ABB RAPID module: d6a8df4c.mod

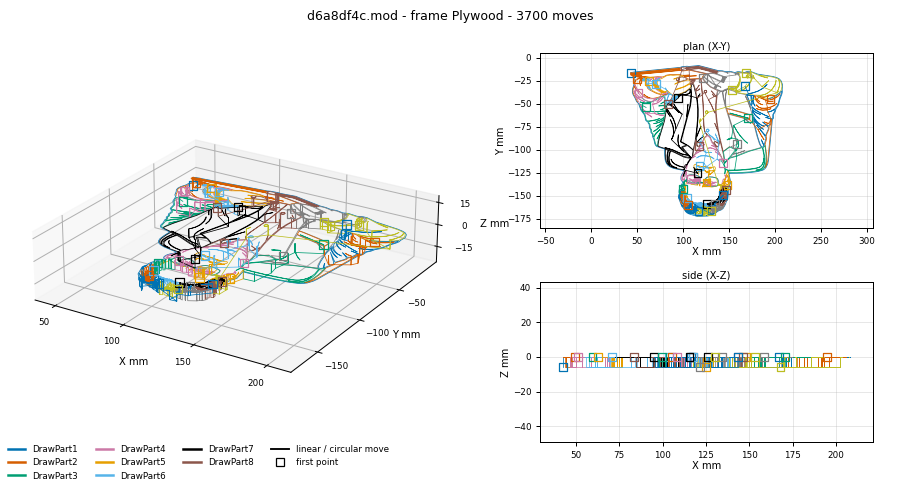
[picture p0: tool path of d6a8df4c.mod in frame Plywood, 3700 of 3702 moves have a stored position in this frame; points joined in program order, loops and branches not executed]
MODULE ImageDraw
  ! Generated 2026-10-07 09:12 for ABB GoFa CRB 15000-5/0.95: 203 strokes
  ! Page 250 x 180 mm. Work object Plywood: Z points DOWN, so pen-up is -Z and the tool uses orientation [1,0,0,0].
  ! Uses the tool 'tcp' and work object 'Plywood' that already exist on the controller.
  CONST robtarget pOrigin:=[[0,0,0],[1,0,0,0],[0,0,0,0],[9E9,9E9,9E9,9E9,9E9,9E9]];
  CONST jointtarget jHome:=[[0,0,0,0,30,0],[9E9,9E9,9E9,9E9,9E9,9E9]];
  CONST speeddata vTravel:=[250,200,5000,1000];

  PROC DrawImage()
    SingArea\Wrist;
    ConfL\Off;
    ConfJ\Off;
    MoveAbsJ jHome\NoEOffs,vTravel,fine,tcp;
    DrawPart1;
    DrawPart2;
    DrawPart3;
    DrawPart4;
    DrawPart5;
    DrawPart6;
    DrawPart7;
    DrawPart8;
    DrawPart9;
    DrawPart10;
    DrawPart11;
    DrawPart12;
    DrawPart13;
    DrawPart14;
    DrawPart15;
    DrawPart16;
    DrawPart17;
    DrawPart18;
    DrawPart19;
    DrawPart20;
    DrawPart21;
    DrawPart22;
    DrawPart23;
    DrawPart24;
    DrawPart25;
    DrawPart26;
    DrawPart27;
    DrawPart28;
    DrawPart29;
    DrawPart30;
    DrawPart31;
    MoveAbsJ jHome\NoEOffs,vTravel,fine,tcp;
  ENDPROC

  PROC DrawPart1()
    MoveL Offs(pOrigin,42.73,-16.05,-6.00),vTravel,z5,tcp\WObj:=Plywood;
    MoveL Offs(pOrigin,42.73,-16.05,-0.00),v60,z0,tcp\WObj:=Plywood;
    MoveL Offs(pOrigin,46.16,-15.41,-0.00),v40,z0,tcp\WObj:=Plywood;
    MoveL Offs(pOrigin,96.63,-10.31,-0.00),v40,z0,tcp\WObj:=Plywood;
    MoveL Offs(pOrigin,98.76,-9.57,-0.00),v40,z0,tcp\WObj:=Plywood;
    MoveL Offs(pOrigin,104.18,-9.04,-0.00),v40,z0,tcp\WObj:=Plywood;
    MoveL Offs(pOrigin,106.09,-9.36,-0.00),v40,z0,tcp\WObj:=Plywood;
    MoveL Offs(pOrigin,116.93,-8.29,-0.00),v40,z0,tcp\WObj:=Plywood;
    MoveL Offs(pOrigin,138.28,-13.82,-0.00),v40,z0,tcp\WObj:=Plywood;
    MoveL Offs(pOrigin,142.64,-14.03,-0.00),v40,z0,tcp\WObj:=Plywood;
    MoveL Offs(pOrigin,146.36,-14.99,-0.00),v40,z0,tcp\WObj:=Plywood;
    MoveL Offs(pOrigin,151.77,-14.77,-0.00),v40,z0,tcp\WObj:=Plywood;
    MoveL Offs(pOrigin,156.24,-15.94,-0.00),v40,z0,tcp\WObj:=Plywood;
    MoveL Offs(pOrigin,159.11,-14.99,-0.00),v40,z0,tcp\WObj:=Plywood;
    MoveL Offs(pOrigin,160.81,-14.99,-0.00),v40,z0,tcp\WObj:=Plywood;
    MoveL Offs(pOrigin,166.54,-15.94,-0.00),v40,z0,tcp\WObj:=Plywood;
    MoveL Offs(pOrigin,170.26,-14.56,-0.00),v40,z0,tcp\WObj:=Plywood;
    MoveL Offs(pOrigin,173.02,-14.56,-0.00),v40,z0,tcp\WObj:=Plywood;
    MoveL Offs(pOrigin,181.10,-17.64,-0.00),v40,z0,tcp\WObj:=Plywood;
    MoveL Offs(pOrigin,197.99,-20.30,-0.00),v40,z0,tcp\WObj:=Plywood;
    MoveL Offs(pOrigin,202.14,-21.54,-0.00),v40,z0,tcp\WObj:=Plywood;
    MoveL Offs(pOrigin,204.79,-22.96,-0.00),v40,z0,tcp\WObj:=Plywood;
    MoveL Offs(pOrigin,206.74,-25.19,-0.00),v40,z0,tcp\WObj:=Plywood;
    MoveL Offs(pOrigin,207.98,-28.59,-0.00),v40,z0,tcp\WObj:=Plywood;
    MoveL Offs(pOrigin,208.19,-30.08,-0.00),v40,z0,tcp\WObj:=Plywood;
    MoveL Offs(pOrigin,207.77,-34.33,-0.00),v40,z0,tcp\WObj:=Plywood;
    MoveL Offs(pOrigin,207.98,-37.09,-0.00),v40,z0,tcp\WObj:=Plywood;
    MoveL Offs(pOrigin,207.38,-39.64,-0.00),v40,z0,tcp\WObj:=Plywood;
    MoveL Offs(pOrigin,205.54,-44.31,-0.00),v40,z0,tcp\WObj:=Plywood;
    MoveL Offs(pOrigin,203.77,-51.01,-0.00),v40,z0,tcp\WObj:=Plywood;
    MoveL Offs(pOrigin,203.06,-52.60,-0.00),v40,z0,tcp\WObj:=Plywood;
    MoveL Offs(pOrigin,201.15,-55.26,-0.00),v40,z0,tcp\WObj:=Plywood;
    MoveL Offs(pOrigin,200.15,-58.66,-0.00),v40,z0,tcp\WObj:=Plywood;
    MoveL Offs(pOrigin,198.49,-61.31,-0.00),v40,z0,tcp\WObj:=Plywood;
    MoveL Offs(pOrigin,198.42,-65.14,-0.00),v40,z0,tcp\WObj:=Plywood;
    MoveL Offs(pOrigin,197.89,-66.31,-0.00),v40,z0,tcp\WObj:=Plywood;
    MoveL Offs(pOrigin,197.14,-66.94,-0.00),v40,z0,tcp\WObj:=Plywood;
    MoveL Offs(pOrigin,192.89,-111.36,-0.00),v40,z0,tcp\WObj:=Plywood;
    MoveL Offs(pOrigin,192.15,-115.18,-0.00),v40,z0,tcp\WObj:=Plywood;
    MoveL Offs(pOrigin,190.45,-119.01,-0.00),v40,z0,tcp\WObj:=Plywood;
    MoveL Offs(pOrigin,188.75,-120.92,-0.00),v40,z0,tcp\WObj:=Plywood;
    MoveL Offs(pOrigin,186.73,-122.23,-0.00),v40,z0,tcp\WObj:=Plywood;
    MoveL Offs(pOrigin,181.10,-123.79,-0.00),v40,z0,tcp\WObj:=Plywood;
    MoveL Offs(pOrigin,173.88,-124.74,-0.00),v40,z0,tcp\WObj:=Plywood;
    MoveL Offs(pOrigin,164.31,-125.49,-0.00),v40,z0,tcp\WObj:=Plywood;
    MoveL Offs(pOrigin,149.76,-125.74,-0.00),v40,z0,tcp\WObj:=Plywood;
    MoveL Offs(pOrigin,151.67,-135.16,-0.00),v40,z0,tcp\WObj:=Plywood;
    MoveL Offs(pOrigin,151.07,-137.60,-0.00),v40,z0,tcp\WObj:=Plywood;
    MoveL Offs(pOrigin,150.00,-139.41,-0.00),v40,z0,tcp\WObj:=Plywood;
    MoveL Offs(pOrigin,150.15,-140.26,-0.00),v40,z0,tcp\WObj:=Plywood;
    MoveL Offs(pOrigin,149.76,-140.79,-0.00),v40,z0,tcp\WObj:=Plywood;
    MoveL Offs(pOrigin,149.44,-143.55,-0.00),v40,z0,tcp\WObj:=Plywood;
    MoveL Offs(pOrigin,149.12,-143.76,-0.00),v40,z0,tcp\WObj:=Plywood;
    MoveL Offs(pOrigin,149.23,-147.27,-0.00),v40,z0,tcp\WObj:=Plywood;
    MoveL Offs(pOrigin,148.23,-154.81,-0.00),v40,z0,tcp\WObj:=Plywood;
    MoveL Offs(pOrigin,147.03,-156.19,-0.00),v40,z0,tcp\WObj:=Plywood;
    MoveL Offs(pOrigin,146.11,-159.38,-0.00),v40,z0,tcp\WObj:=Plywood;
    MoveL Offs(pOrigin,143.49,-163.95,-0.00),v40,z0,tcp\WObj:=Plywood;
    MoveL Offs(pOrigin,141.57,-165.47,-0.00),v40,z0,tcp\WObj:=Plywood;
    MoveL Offs(pOrigin,137.86,-166.89,-0.00),v40,z0,tcp\WObj:=Plywood;
    MoveL Offs(pOrigin,134.14,-169.83,-0.00),v40,z0,tcp\WObj:=Plywood;
    MoveL Offs(pOrigin,132.12,-170.75,-0.00),v40,z0,tcp\WObj:=Plywood;
    MoveL Offs(pOrigin,126.38,-172.24,-0.00),v40,z0,tcp\WObj:=Plywood;
    MoveL Offs(pOrigin,115.22,-172.56,-0.00),v40,z0,tcp\WObj:=Plywood;
    MoveL Offs(pOrigin,106.41,-169.94,-0.00),v40,z0,tcp\WObj:=Plywood;
    MoveL Offs(pOrigin,104.18,-168.84,-0.00),v40,z0,tcp\WObj:=Plywood;
    MoveL Offs(pOrigin,102.58,-167.35,-0.00),v40,z0,tcp\WObj:=Plywood;
    MoveL Offs(pOrigin,100.67,-164.06,-0.00),v40,z0,tcp\WObj:=Plywood;
    MoveL Offs(pOrigin,98.30,-161.40,-0.00),v40,z0,tcp\WObj:=Plywood;
    MoveL Offs(pOrigin,94.72,-151.73,-0.00),v40,z0,tcp\WObj:=Plywood;
    MoveL Offs(pOrigin,94.93,-149.61,-0.00),v40,z0,tcp\WObj:=Plywood;
    MoveL Offs(pOrigin,95.75,-147.80,-0.00),v40,z0,tcp\WObj:=Plywood;
    MoveL Offs(pOrigin,95.36,-146.21,-0.00),v40,z0,tcp\WObj:=Plywood;
    MoveL Offs(pOrigin,95.57,-143.76,-0.00),v40,z0,tcp\WObj:=Plywood;
    MoveL Offs(pOrigin,96.60,-140.68,-0.00),v40,z0,tcp\WObj:=Plywood;
    MoveL Offs(pOrigin,99.50,-135.58,-0.00),v40,z0,tcp\WObj:=Plywood;
    MoveL Offs(pOrigin,99.50,-134.73,-0.00),v40,z0,tcp\WObj:=Plywood;
    MoveL Offs(pOrigin,98.65,-134.31,-0.00),v40,z0,tcp\WObj:=Plywood;
    MoveL Offs(pOrigin,97.80,-133.14,-0.00),v40,z0,tcp\WObj:=Plywood;
    MoveL Offs(pOrigin,97.48,-131.76,-0.00),v40,z0,tcp\WObj:=Plywood;
    MoveL Offs(pOrigin,97.59,-129.10,-0.00),v40,z0,tcp\WObj:=Plywood;
    MoveL Offs(pOrigin,98.19,-127.51,-0.00),v40,z0,tcp\WObj:=Plywood;
    MoveL Offs(pOrigin,99.68,-125.17,-0.00),v40,z0,tcp\WObj:=Plywood;
    MoveL Offs(pOrigin,100.53,-122.72,-0.00),v40,z0,tcp\WObj:=Plywood;
    MoveL Offs(pOrigin,89.51,-120.28,-0.00),v40,z0,tcp\WObj:=Plywood;
    MoveL Offs(pOrigin,85.58,-118.62,-0.00),v40,z0,tcp\WObj:=Plywood;
    MoveL Offs(pOrigin,83.46,-117.09,-0.00),v40,z0,tcp\WObj:=Plywood;
    MoveL Offs(pOrigin,81.61,-114.76,-0.00),v40,z0,tcp\WObj:=Plywood;
    MoveL Offs(pOrigin,80.38,-111.46,-0.00),v40,z0,tcp\WObj:=Plywood;
    MoveL Offs(pOrigin,79.84,-106.26,-0.00),v40,z0,tcp\WObj:=Plywood;
    MoveL Offs(pOrigin,79.77,-99.24,-0.00),v40,z0,tcp\WObj:=Plywood;
    MoveL Offs(pOrigin,71.66,-96.62,-0.00),v40,z0,tcp\WObj:=Plywood;
    MoveL Offs(pOrigin,70.71,-96.06,-0.00),v40,z0,tcp\WObj:=Plywood;
    MoveL Offs(pOrigin,69.61,-94.68,-0.00),v40,z0,tcp\WObj:=Plywood;
    MoveL Offs(pOrigin,68.90,-92.97,-0.00),v40,z0,tcp\WObj:=Plywood;
    MoveL Offs(pOrigin,68.16,-89.26,-0.00),v40,z0,tcp\WObj:=Plywood;
    MoveL Offs(pOrigin,66.56,-85.43,-0.00),v40,z0,tcp\WObj:=Plywood;
    MoveL Offs(pOrigin,66.39,-82.99,-0.00),v40,z0,tcp\WObj:=Plywood;
    MoveL Offs(pOrigin,64.86,-81.07,-0.00),v40,z0,tcp\WObj:=Plywood;
    MoveL Offs(pOrigin,64.69,-77.99,-0.00),v40,z0,tcp\WObj:=Plywood;
    MoveL Offs(pOrigin,63.69,-76.93,-0.00),v40,z0,tcp\WObj:=Plywood;
    MoveL Offs(pOrigin,63.16,-75.76,-0.00),v40,z0,tcp\WObj:=Plywood;
    MoveL Offs(pOrigin,62.99,-72.47,-0.00),v40,z0,tcp\WObj:=Plywood;
    MoveL Offs(pOrigin,61.82,-70.88,-0.00),v40,z0,tcp\WObj:=Plywood;
    MoveL Offs(pOrigin,61.46,-69.39,-0.00),v40,z0,tcp\WObj:=Plywood;
    MoveL Offs(pOrigin,60.19,-69.00,-0.00),v40,z0,tcp\WObj:=Plywood;
    MoveL Offs(pOrigin,59.20,-68.01,-0.00),v40,z0,tcp\WObj:=Plywood;
    MoveL Offs(pOrigin,57.89,-62.27,-0.00),v40,z0,tcp\WObj:=Plywood;
    MoveL Offs(pOrigin,53.88,-56.85,-0.00),v40,z0,tcp\WObj:=Plywood;
    MoveL Offs(pOrigin,51.33,-49.62,-0.00),v40,z0,tcp\WObj:=Plywood;
    MoveL Offs(pOrigin,49.78,-48.24,-0.00),v40,z0,tcp\WObj:=Plywood;
    MoveL Offs(pOrigin,49.00,-47.08,-0.00),v40,z0,tcp\WObj:=Plywood;
    MoveL Offs(pOrigin,47.15,-42.93,-0.00),v40,z0,tcp\WObj:=Plywood;
    MoveL Offs(pOrigin,45.49,-40.17,-0.00),v40,z0,tcp\WObj:=Plywood;
    MoveL Offs(pOrigin,44.67,-37.51,-0.00),v40,z0,tcp\WObj:=Plywood;
    MoveL Offs(pOrigin,44.78,-34.11,-0.00),v40,z0,tcp\WObj:=Plywood;
    MoveL Offs(pOrigin,46.27,-29.23,-0.00),v40,z0,tcp\WObj:=Plywood;
    MoveL Offs(pOrigin,46.16,-27.42,-0.00),v40,z0,tcp\WObj:=Plywood;
    MoveL Offs(pOrigin,46.66,-25.51,-0.00),v40,z0,tcp\WObj:=Plywood;
    MoveL Offs(pOrigin,48.08,-23.81,-0.00),v40,z0,tcp\WObj:=Plywood;
  ENDPROC

  PROC DrawPart2()
    MoveL Offs(pOrigin,49.56,-22.89,-0.00),v40,z0,tcp\WObj:=Plywood;
    MoveL Offs(pOrigin,54.10,-21.68,-0.00),v40,z0,tcp\WObj:=Plywood;
    MoveL Offs(pOrigin,43.29,-19.06,-0.00),v40,z0,tcp\WObj:=Plywood;
    MoveL Offs(pOrigin,42.55,-18.17,-0.00),v40,z0,tcp\WObj:=Plywood;
    MoveL Offs(pOrigin,42.73,-16.05,-0.00),v40,z0,tcp\WObj:=Plywood;
    MoveL Offs(pOrigin,43.51,-16.40,-0.00),v40,z0,tcp\WObj:=Plywood;
    MoveL Offs(pOrigin,43.22,-17.01,-0.00),v40,z0,tcp\WObj:=Plywood;
    MoveL Offs(pOrigin,43.61,-17.22,-0.00),v40,z0,tcp\WObj:=Plywood;
    MoveL Offs(pOrigin,95.57,-11.91,-0.00),v40,z0,tcp\WObj:=Plywood;
    MoveL Offs(pOrigin,96.53,-11.69,-0.00),v40,z0,tcp\WObj:=Plywood;
    MoveL Offs(pOrigin,96.63,-11.16,-0.00),v40,z0,tcp\WObj:=Plywood;
    MoveL Offs(pOrigin,95.04,-11.06,-0.00),v40,z0,tcp\WObj:=Plywood;
    MoveL Offs(pOrigin,43.51,-16.40,-0.00),v40,z0,tcp\WObj:=Plywood;
    MoveL Offs(pOrigin,43.72,-17.54,-0.00),v40,z0,tcp\WObj:=Plywood;
    MoveL Offs(pOrigin,43.29,-18.07,-0.00),v40,z0,tcp\WObj:=Plywood;
    MoveL Offs(pOrigin,44.89,-18.28,-0.00),v40,z0,tcp\WObj:=Plywood;
    MoveL Offs(pOrigin,93.12,-13.71,-0.00),v40,z0,tcp\WObj:=Plywood;
    MoveL Offs(pOrigin,96.95,-13.07,-0.00),v40,z0,tcp\WObj:=Plywood;
    MoveL Offs(pOrigin,96.31,-12.23,-0.00),v40,z0,tcp\WObj:=Plywood;
    MoveL Offs(pOrigin,43.72,-17.54,-0.00),v40,fine,tcp\WObj:=Plywood;
    MoveL Offs(pOrigin,43.72,-17.54,-6.00),v60,z5,tcp\WObj:=Plywood;
    MoveL Offs(pOrigin,44.50,-18.81,-6.00),vTravel,z5,tcp\WObj:=Plywood;
    MoveL Offs(pOrigin,44.50,-18.81,-0.00),v60,z0,tcp\WObj:=Plywood;
    MoveL Offs(pOrigin,53.17,-20.94,-0.00),v40,z0,tcp\WObj:=Plywood;
    MoveL Offs(pOrigin,63.16,-22.11,-0.00),v40,z0,tcp\WObj:=Plywood;
    MoveL Offs(pOrigin,65.11,-21.58,-0.00),v40,z0,tcp\WObj:=Plywood;
    MoveL Offs(pOrigin,49.53,-19.45,-0.00),v40,z0,tcp\WObj:=Plywood;
    MoveL Offs(pOrigin,64.22,-21.15,-0.00),v40,z0,tcp\WObj:=Plywood;
    MoveL Offs(pOrigin,72.41,-20.41,-0.00),v40,z0,tcp\WObj:=Plywood;
    MoveL Offs(pOrigin,77.40,-20.73,-0.00),v40,z0,tcp\WObj:=Plywood;
    MoveL Offs(pOrigin,78.68,-20.44,-0.00),v40,z0,tcp\WObj:=Plywood;
    MoveL Offs(pOrigin,82.07,-18.71,-0.00),v40,z0,tcp\WObj:=Plywood;
    MoveL Offs(pOrigin,85.69,-18.17,-0.00),v40,z0,tcp\WObj:=Plywood;
    MoveL Offs(pOrigin,95.99,-18.17,-0.00),v40,z0,tcp\WObj:=Plywood;
    MoveL Offs(pOrigin,99.50,-18.95,-0.00),v40,z0,tcp\WObj:=Plywood;
    MoveL Offs(pOrigin,106.87,-18.71,-0.00),v40,z0,tcp\WObj:=Plywood;
    MoveL Offs(pOrigin,100.14,-19.24,-0.00),v40,z0,tcp\WObj:=Plywood;
    MoveL Offs(pOrigin,100.88,-19.98,-0.00),v40,z0,tcp\WObj:=Plywood;
    MoveL Offs(pOrigin,114.41,-19.45,-0.00),v40,z0,tcp\WObj:=Plywood;
    MoveL Offs(pOrigin,101.13,-20.30,-0.00),v40,z0,tcp\WObj:=Plywood;
    MoveL Offs(pOrigin,103.86,-21.89,-0.00),v40,z0,tcp\WObj:=Plywood;
    MoveL Offs(pOrigin,105.03,-23.03,-0.00),v40,z0,tcp\WObj:=Plywood;
    MoveL Offs(pOrigin,120.32,-22.11,-0.00),v40,z0,tcp\WObj:=Plywood;
    MoveL Offs(pOrigin,120.75,-21.89,-0.00),v40,z0,tcp\WObj:=Plywood;
    MoveL Offs(pOrigin,120.93,-20.41,-0.00),v40,z0,tcp\WObj:=Plywood;
    MoveL Offs(pOrigin,121.99,-19.45,-0.00),v40,z0,tcp\WObj:=Plywood;
    MoveL Offs(pOrigin,122.59,-18.07,-0.00),v40,z0,tcp\WObj:=Plywood;
    MoveL Offs(pOrigin,124.72,-17.33,-0.00),v40,z0,tcp\WObj:=Plywood;
    MoveL Offs(pOrigin,105.98,-13.18,-0.00),v40,z0,tcp\WObj:=Plywood;
    MoveL Offs(pOrigin,104.49,-13.71,-0.00),v40,z0,tcp\WObj:=Plywood;
    MoveL Offs(pOrigin,99.18,-14.24,-0.00),v40,z0,tcp\WObj:=Plywood;
    MoveL Offs(pOrigin,98.12,-14.14,-0.00),v40,z0,tcp\WObj:=Plywood;
    MoveL Offs(pOrigin,97.16,-13.61,-0.00),v40,z0,tcp\WObj:=Plywood;
    MoveL Offs(pOrigin,45.53,-18.49,-0.00),v40,z0,tcp\WObj:=Plywood;
    MoveL Offs(pOrigin,44.50,-18.81,-0.00),v40,fine,tcp\WObj:=Plywood;
    MoveL Offs(pOrigin,44.50,-18.81,-6.00),v60,z5,tcp\WObj:=Plywood;
    MoveL Offs(pOrigin,47.97,-24.87,-6.00),vTravel,z5,tcp\WObj:=Plywood;
    MoveL Offs(pOrigin,47.97,-24.87,-0.00),v60,z0,tcp\WObj:=Plywood;
    MoveL Offs(pOrigin,47.12,-26.36,-0.00),v40,z0,tcp\WObj:=Plywood;
    MoveL Offs(pOrigin,47.51,-29.23,-0.00),v40,z0,tcp\WObj:=Plywood;
    MoveL Offs(pOrigin,49.99,-34.54,-0.00),v40,z0,tcp\WObj:=Plywood;
    MoveL Offs(pOrigin,53.00,-37.30,-0.00),v40,z0,tcp\WObj:=Plywood;
    MoveL Offs(pOrigin,57.00,-41.76,-0.00),v40,z0,tcp\WObj:=Plywood;
    MoveL Offs(pOrigin,58.59,-42.75,-0.00),v40,z0,tcp\WObj:=Plywood;
    MoveL Offs(pOrigin,61.14,-43.67,-0.00),v40,z0,tcp\WObj:=Plywood;
    MoveL Offs(pOrigin,63.73,-43.89,-0.00),v40,z0,tcp\WObj:=Plywood;
    MoveL Offs(pOrigin,59.87,-42.01,-0.00),v40,z0,tcp\WObj:=Plywood;
    MoveL Offs(pOrigin,57.07,-39.67,-0.00),v40,z0,tcp\WObj:=Plywood;
    MoveL Offs(pOrigin,60.29,-42.01,-0.00),v40,z0,tcp\WObj:=Plywood;
    MoveL Offs(pOrigin,62.95,-43.29,-0.00),v40,z0,tcp\WObj:=Plywood;
    MoveL Offs(pOrigin,65.71,-43.99,-0.00),v40,z0,tcp\WObj:=Plywood;
    MoveL Offs(pOrigin,67.94,-43.99,-0.00),v40,z0,tcp\WObj:=Plywood;
    MoveL Offs(pOrigin,72.30,-43.04,-0.00),v40,z0,tcp\WObj:=Plywood;
    MoveL Offs(pOrigin,82.39,-39.67,-0.00),v40,z0,tcp\WObj:=Plywood;
    MoveL Offs(pOrigin,85.01,-38.36,-0.00),v40,z0,tcp\WObj:=Plywood;
    MoveL Offs(pOrigin,84.41,-37.87,-0.00),v40,z0,tcp\WObj:=Plywood;
    MoveL Offs(pOrigin,82.29,-39.14,-0.00),v40,z0,tcp\WObj:=Plywood;
    MoveL Offs(pOrigin,80.48,-39.74,-0.00),v40,z0,tcp\WObj:=Plywood;
    MoveL Offs(pOrigin,78.57,-40.06,-0.00),v40,z0,tcp\WObj:=Plywood;
    MoveL Offs(pOrigin,75.91,-39.96,-0.00),v40,z0,tcp\WObj:=Plywood;
    MoveL Offs(pOrigin,72.62,-39.21,-0.00),v40,z0,tcp\WObj:=Plywood;
    MoveL Offs(pOrigin,69.86,-38.19,-0.00),v40,z0,tcp\WObj:=Plywood;
    MoveL Offs(pOrigin,63.59,-35.00,-0.00),v40,z0,tcp\WObj:=Plywood;
    MoveL Offs(pOrigin,61.46,-33.26,-0.00),v40,z0,tcp\WObj:=Plywood;
    MoveL Offs(pOrigin,60.29,-30.82,-0.00),v40,z0,tcp\WObj:=Plywood;
    MoveL Offs(pOrigin,59.76,-27.95,-0.00),v40,z0,tcp\WObj:=Plywood;
    MoveL Offs(pOrigin,59.76,-25.51,-0.00),v40,z0,tcp\WObj:=Plywood;
    MoveL Offs(pOrigin,60.40,-22.64,-0.00),v40,z0,tcp\WObj:=Plywood;
    MoveL Offs(pOrigin,60.08,-22.32,-0.00),v40,z0,tcp\WObj:=Plywood;
    MoveL Offs(pOrigin,59.16,-22.42,-0.00),v40,z0,tcp\WObj:=Plywood;
    MoveL Offs(pOrigin,58.63,-23.91,-0.00),v40,z0,tcp\WObj:=Plywood;
    MoveL Offs(pOrigin,57.74,-24.90,-0.00),v40,z0,tcp\WObj:=Plywood;
    MoveL Offs(pOrigin,57.11,-24.69,-0.00),v40,z0,tcp\WObj:=Plywood;
    MoveL Offs(pOrigin,56.58,-25.08,-0.00),v40,z0,tcp\WObj:=Plywood;
    MoveL Offs(pOrigin,55.34,-24.98,-0.00),v40,z0,tcp\WObj:=Plywood;
    MoveL Offs(pOrigin,55.30,-23.91,-0.00),v40,z0,tcp\WObj:=Plywood;
    MoveL Offs(pOrigin,56.22,-22.42,-0.00),v40,z0,tcp\WObj:=Plywood;
    MoveL Offs(pOrigin,56.04,-22.21,-0.00),v40,z0,tcp\WObj:=Plywood;
    MoveL Offs(pOrigin,55.09,-22.57,-0.00),v40,z0,tcp\WObj:=Plywood;
    MoveL Offs(pOrigin,53.71,-23.70,-0.00),v40,z0,tcp\WObj:=Plywood;
    MoveL Offs(pOrigin,52.75,-26.46,-0.00),v40,z0,tcp\WObj:=Plywood;
    MoveL Offs(pOrigin,53.56,-30.32,-0.00),v40,z0,tcp\WObj:=Plywood;
    MoveL Offs(pOrigin,52.54,-27.74,-0.00),v40,z0,tcp\WObj:=Plywood;
    MoveL Offs(pOrigin,52.43,-25.51,-0.00),v40,z0,tcp\WObj:=Plywood;
    MoveL Offs(pOrigin,53.60,-22.57,-0.00),v40,z0,tcp\WObj:=Plywood;
    MoveL Offs(pOrigin,51.16,-22.96,-0.00),v40,z0,tcp\WObj:=Plywood;
    MoveL Offs(pOrigin,49.67,-23.56,-0.00),v40,z0,tcp\WObj:=Plywood;
    MoveL Offs(pOrigin,47.97,-24.87,-0.00),v40,fine,tcp\WObj:=Plywood;
    MoveL Offs(pOrigin,47.97,-24.87,-6.00),v60,z5,tcp\WObj:=Plywood;
    MoveL Offs(pOrigin,47.01,-28.98,-6.00),vTravel,z5,tcp\WObj:=Plywood;
    MoveL Offs(pOrigin,47.01,-28.98,-0.00),v60,z0,tcp\WObj:=Plywood;
    MoveL Offs(pOrigin,47.33,-31.14,-0.00),v40,z0,tcp\WObj:=Plywood;
    MoveL Offs(pOrigin,49.31,-35.95,-0.00),v40,z0,tcp\WObj:=Plywood;
    MoveL Offs(pOrigin,46.48,-30.82,-0.00),v40,z0,tcp\WObj:=Plywood;
    MoveL Offs(pOrigin,45.31,-35.28,-0.00),v40,z0,tcp\WObj:=Plywood;
    MoveL Offs(pOrigin,45.42,-37.72,-0.00),v40,z0,tcp\WObj:=Plywood;
    MoveL Offs(pOrigin,46.02,-39.64,-0.00),v40,z0,tcp\WObj:=Plywood;
    MoveL Offs(pOrigin,48.22,-43.36,-0.00),v40,z0,tcp\WObj:=Plywood;
    MoveL Offs(pOrigin,49.63,-46.76,-0.00),v40,z0,tcp\WObj:=Plywood;
    MoveL Offs(pOrigin,50.52,-47.92,-0.00),v40,z0,tcp\WObj:=Plywood;
  ENDPROC

  PROC DrawPart3()
    MoveL Offs(pOrigin,59.59,-53.95,-0.00),v40,z0,tcp\WObj:=Plywood;
    MoveL Offs(pOrigin,52.43,-50.19,-0.00),v40,z0,tcp\WObj:=Plywood;
    MoveL Offs(pOrigin,53.67,-54.51,-0.00),v40,z0,tcp\WObj:=Plywood;
    MoveL Offs(pOrigin,54.63,-56.64,-0.00),v40,z0,tcp\WObj:=Plywood;
    MoveL Offs(pOrigin,58.42,-61.74,-0.00),v40,z0,tcp\WObj:=Plywood;
    MoveL Offs(pOrigin,59.55,-66.84,-0.00),v40,z0,tcp\WObj:=Plywood;
    MoveL Offs(pOrigin,60.19,-68.11,-0.00),v40,z0,tcp\WObj:=Plywood;
    MoveL Offs(pOrigin,61.36,-68.64,-0.00),v40,z0,tcp\WObj:=Plywood;
    MoveL Offs(pOrigin,65.29,-68.32,-0.00),v40,z0,tcp\WObj:=Plywood;
    MoveL Offs(pOrigin,69.96,-67.37,-0.00),v40,z0,tcp\WObj:=Plywood;
    MoveL Offs(pOrigin,74.78,-65.92,-0.00),v40,z0,tcp\WObj:=Plywood;
    MoveL Offs(pOrigin,70.28,-67.69,-0.00),v40,z0,tcp\WObj:=Plywood;
    MoveL Offs(pOrigin,62.74,-69.18,-0.00),v40,z0,tcp\WObj:=Plywood;
    MoveL Offs(pOrigin,62.31,-69.49,-0.00),v40,z0,tcp\WObj:=Plywood;
    MoveL Offs(pOrigin,62.49,-70.56,-0.00),v40,z0,tcp\WObj:=Plywood;
    MoveL Offs(pOrigin,63.80,-72.47,-0.00),v40,z0,tcp\WObj:=Plywood;
    MoveL Offs(pOrigin,64.05,-76.08,-0.00),v40,z0,tcp\WObj:=Plywood;
    MoveL Offs(pOrigin,65.50,-78.21,-0.00),v40,z0,tcp\WObj:=Plywood;
    MoveL Offs(pOrigin,65.64,-81.07,-0.00),v40,z0,tcp\WObj:=Plywood;
    MoveL Offs(pOrigin,66.88,-82.24,-0.00),v40,z0,tcp\WObj:=Plywood;
    MoveL Offs(pOrigin,67.20,-82.99,-0.00),v40,z0,tcp\WObj:=Plywood;
    MoveL Offs(pOrigin,67.09,-84.47,-0.00),v40,z0,tcp\WObj:=Plywood;
    MoveL Offs(pOrigin,67.52,-85.82,-0.00),v40,z0,tcp\WObj:=Plywood;
    MoveL Offs(pOrigin,70.18,-81.93,-0.00),v40,z0,tcp\WObj:=Plywood;
    MoveL Offs(pOrigin,74.78,-77.85,-0.00),v40,z0,tcp\WObj:=Plywood;
    MoveL Offs(pOrigin,69.75,-83.52,-0.00),v40,z0,tcp\WObj:=Plywood;
    MoveL Offs(pOrigin,68.76,-85.01,-0.00),v40,z0,tcp\WObj:=Plywood;
    MoveL Offs(pOrigin,68.09,-86.81,-0.00),v40,z0,tcp\WObj:=Plywood;
    MoveL Offs(pOrigin,69.93,-93.72,-0.00),v40,z0,tcp\WObj:=Plywood;
    MoveL Offs(pOrigin,70.71,-94.99,-0.00),v40,z0,tcp\WObj:=Plywood;
    MoveL Offs(pOrigin,72.19,-96.02,-0.00),v40,z0,tcp\WObj:=Plywood;
    MoveL Offs(pOrigin,72.41,-91.28,-0.00),v40,z0,tcp\WObj:=Plywood;
    MoveL Offs(pOrigin,74.81,-82.46,-0.00),v40,z0,tcp\WObj:=Plywood;
    MoveL Offs(pOrigin,73.54,-84.26,-0.00),v40,z0,tcp\WObj:=Plywood;
    MoveL Offs(pOrigin,71.49,-88.30,-0.00),v40,z0,tcp\WObj:=Plywood;
    MoveL Offs(pOrigin,75.42,-80.44,-0.00),v40,z0,tcp\WObj:=Plywood;
    MoveL Offs(pOrigin,78.36,-70.80,-0.00),v40,z0,tcp\WObj:=Plywood;
    MoveL Offs(pOrigin,74.64,-75.12,-0.00),v40,z0,tcp\WObj:=Plywood;
    MoveL Offs(pOrigin,71.88,-77.78,-0.00),v40,z0,tcp\WObj:=Plywood;
    MoveL Offs(pOrigin,69.32,-79.52,-0.00),v40,z0,tcp\WObj:=Plywood;
    MoveL Offs(pOrigin,67.59,-80.01,-0.00),v40,z0,tcp\WObj:=Plywood;
    MoveL Offs(pOrigin,71.56,-77.25,-0.00),v40,z0,tcp\WObj:=Plywood;
    MoveL Offs(pOrigin,75.59,-73.00,-0.00),v40,z0,tcp\WObj:=Plywood;
    MoveL Offs(pOrigin,77.47,-70.56,-0.00),v40,z0,tcp\WObj:=Plywood;
    MoveL Offs(pOrigin,74.00,-73.04,-0.00),v40,z0,tcp\WObj:=Plywood;
    MoveL Offs(pOrigin,70.46,-74.81,-0.00),v40,z0,tcp\WObj:=Plywood;
    MoveL Offs(pOrigin,73.26,-73.25,-0.00),v40,z0,tcp\WObj:=Plywood;
    MoveL Offs(pOrigin,77.19,-70.34,-0.00),v40,z0,tcp\WObj:=Plywood;
    MoveL Offs(pOrigin,78.96,-68.43,-0.00),v40,z0,tcp\WObj:=Plywood;
    MoveL Offs(pOrigin,79.24,-67.16,-0.00),v40,z0,tcp\WObj:=Plywood;
    MoveL Offs(pOrigin,76.87,-68.79,-0.00),v40,z0,tcp\WObj:=Plywood;
    MoveL Offs(pOrigin,73.89,-70.27,-0.00),v40,z0,tcp\WObj:=Plywood;
    MoveL Offs(pOrigin,70.07,-71.30,-0.00),v40,z0,tcp\WObj:=Plywood;
    MoveL Offs(pOrigin,67.80,-71.41,-0.00),v40,z0,tcp\WObj:=Plywood;
    MoveL Offs(pOrigin,71.34,-70.77,-0.00),v40,z0,tcp\WObj:=Plywood;
    MoveL Offs(pOrigin,74.43,-69.64,-0.00),v40,z0,tcp\WObj:=Plywood;
    MoveL Offs(pOrigin,77.51,-67.79,-0.00),v40,z0,tcp\WObj:=Plywood;
    MoveL Offs(pOrigin,79.49,-65.78,-0.00),v40,z0,tcp\WObj:=Plywood;
    MoveL Offs(pOrigin,79.42,-64.89,-0.00),v40,z0,tcp\WObj:=Plywood;
    MoveL Offs(pOrigin,77.08,-66.66,-0.00),v40,z0,tcp\WObj:=Plywood;
    MoveL Offs(pOrigin,74.64,-67.94,-0.00),v40,z0,tcp\WObj:=Plywood;
    MoveL Offs(pOrigin,70.35,-69.28,-0.00),v40,z0,tcp\WObj:=Plywood;
    MoveL Offs(pOrigin,74.21,-67.83,-0.00),v40,z0,tcp\WObj:=Plywood;
    MoveL Offs(pOrigin,78.25,-65.24,-0.00),v40,z0,tcp\WObj:=Plywood;
    MoveL Offs(pOrigin,79.95,-63.12,-0.00),v40,z0,tcp\WObj:=Plywood;
    MoveL Offs(pOrigin,80.27,-60.18,-0.00),v40,z0,tcp\WObj:=Plywood;
    MoveL Offs(pOrigin,78.14,-60.99,-0.00),v40,z0,tcp\WObj:=Plywood;
    MoveL Offs(pOrigin,76.02,-61.10,-0.00),v40,z0,tcp\WObj:=Plywood;
    MoveL Offs(pOrigin,72.05,-60.04,-0.00),v40,z0,tcp\WObj:=Plywood;
    MoveL Offs(pOrigin,74.85,-60.57,-0.00),v40,z0,tcp\WObj:=Plywood;
    MoveL Offs(pOrigin,77.51,-60.57,-0.00),v40,z0,tcp\WObj:=Plywood;
    MoveL Offs(pOrigin,79.74,-59.61,-0.00),v40,z0,tcp\WObj:=Plywood;
    MoveL Offs(pOrigin,80.59,-58.23,-0.00),v40,z0,tcp\WObj:=Plywood;
    MoveL Offs(pOrigin,80.38,-57.98,-0.00),v40,z0,tcp\WObj:=Plywood;
    MoveL Offs(pOrigin,78.25,-58.02,-0.00),v40,z0,tcp\WObj:=Plywood;
    MoveL Offs(pOrigin,72.83,-58.66,-0.00),v40,z0,tcp\WObj:=Plywood;
    MoveL Offs(pOrigin,67.31,-58.76,-0.00),v40,z0,tcp\WObj:=Plywood;
    MoveL Offs(pOrigin,63.02,-58.12,-0.00),v40,z0,tcp\WObj:=Plywood;
    MoveL Offs(pOrigin,70.60,-58.44,-0.00),v40,z0,tcp\WObj:=Plywood;
    MoveL Offs(pOrigin,77.82,-57.70,-0.00),v40,z0,tcp\WObj:=Plywood;
    MoveL Offs(pOrigin,80.59,-57.81,-0.00),v40,z0,tcp\WObj:=Plywood;
    MoveL Offs(pOrigin,80.91,-54.51,-0.00),v40,z0,tcp\WObj:=Plywood;
    MoveL Offs(pOrigin,79.10,-55.50,-0.00),v40,z0,tcp\WObj:=Plywood;
    MoveL Offs(pOrigin,75.35,-56.39,-0.00),v40,z0,tcp\WObj:=Plywood;
    MoveL Offs(pOrigin,77.72,-55.61,-0.00),v40,z0,tcp\WObj:=Plywood;
    MoveL Offs(pOrigin,79.95,-54.41,-0.00),v40,z0,tcp\WObj:=Plywood;
    MoveL Offs(pOrigin,81.01,-53.24,-0.00),v40,z0,tcp\WObj:=Plywood;
    MoveL Offs(pOrigin,80.48,-52.60,-0.00),v40,z0,tcp\WObj:=Plywood;
    MoveL Offs(pOrigin,78.68,-52.07,-0.00),v40,z0,tcp\WObj:=Plywood;
    MoveL Offs(pOrigin,73.29,-52.32,-0.00),v40,z0,tcp\WObj:=Plywood;
    MoveL Offs(pOrigin,76.55,-51.75,-0.00),v40,z0,tcp\WObj:=Plywood;
    MoveL Offs(pOrigin,79.21,-51.75,-0.00),v40,z0,tcp\WObj:=Plywood;
    MoveL Offs(pOrigin,80.59,-52.28,-0.00),v40,z0,tcp\WObj:=Plywood;
    MoveL Offs(pOrigin,81.01,-52.99,-0.00),v40,z0,tcp\WObj:=Plywood;
    MoveL Offs(pOrigin,81.30,-52.81,-0.00),v40,z0,tcp\WObj:=Plywood;
    MoveL Offs(pOrigin,81.15,-50.58,-0.00),v40,z0,tcp\WObj:=Plywood;
    MoveL Offs(pOrigin,80.27,-49.20,-0.00),v40,z0,tcp\WObj:=Plywood;
    MoveL Offs(pOrigin,79.21,-48.42,-0.00),v40,z0,tcp\WObj:=Plywood;
    MoveL Offs(pOrigin,77.82,-48.74,-0.00),v40,z0,tcp\WObj:=Plywood;
    MoveL Offs(pOrigin,75.56,-50.01,-0.00),v40,z0,tcp\WObj:=Plywood;
    MoveL Offs(pOrigin,78.04,-48.21,-0.00),v40,z0,tcp\WObj:=Plywood;
    MoveL Offs(pOrigin,78.89,-47.92,-0.00),v40,z0,tcp\WObj:=Plywood;
    MoveL Offs(pOrigin,80.23,-48.14,-0.00),v40,z0,tcp\WObj:=Plywood;
    MoveL Offs(pOrigin,80.16,-45.48,-0.00),v40,z0,tcp\WObj:=Plywood;
    MoveL Offs(pOrigin,79.45,-42.29,-0.00),v40,z0,tcp\WObj:=Plywood;
    MoveL Offs(pOrigin,78.89,-41.48,-0.00),v40,z0,tcp\WObj:=Plywood;
    MoveL Offs(pOrigin,74.85,-42.79,-0.00),v40,z0,tcp\WObj:=Plywood;
    MoveL Offs(pOrigin,68.47,-46.79,-0.00),v40,z0,tcp\WObj:=Plywood;
    MoveL Offs(pOrigin,63.48,-48.88,-0.00),v40,z0,tcp\WObj:=Plywood;
    MoveL Offs(pOrigin,58.81,-49.52,-0.00),v40,z0,tcp\WObj:=Plywood;
    MoveL Offs(pOrigin,54.34,-48.60,-0.00),v40,z0,tcp\WObj:=Plywood;
    MoveL Offs(pOrigin,53.03,-47.85,-0.00),v40,z0,tcp\WObj:=Plywood;
    MoveL Offs(pOrigin,57.21,-48.88,-0.00),v40,z0,tcp\WObj:=Plywood;
    MoveL Offs(pOrigin,60.29,-48.88,-0.00),v40,z0,tcp\WObj:=Plywood;
    MoveL Offs(pOrigin,63.06,-48.35,-0.00),v40,z0,tcp\WObj:=Plywood;
    MoveL Offs(pOrigin,65.22,-47.39,-0.00),v40,z0,tcp\WObj:=Plywood;
    MoveL Offs(pOrigin,62.21,-47.50,-0.00),v40,z0,tcp\WObj:=Plywood;
    MoveL Offs(pOrigin,60.19,-47.00,-0.00),v40,z0,tcp\WObj:=Plywood;
    MoveL Offs(pOrigin,57.96,-45.94,-0.00),v40,z0,tcp\WObj:=Plywood;
    MoveL Offs(pOrigin,55.09,-43.67,-0.00),v40,z0,tcp\WObj:=Plywood;
  ENDPROC

  PROC DrawPart4()
    MoveL Offs(pOrigin,51.33,-38.58,-0.00),v40,z0,tcp\WObj:=Plywood;
    MoveL Offs(pOrigin,47.01,-28.98,-0.00),v40,fine,tcp\WObj:=Plywood;
    MoveL Offs(pOrigin,47.01,-28.98,-6.00),v60,z5,tcp\WObj:=Plywood;
    MoveL Offs(pOrigin,50.13,-34.96,-6.00),vTravel,z5,tcp\WObj:=Plywood;
    MoveL Offs(pOrigin,50.13,-34.96,-0.00),v60,z0,tcp\WObj:=Plywood;
    MoveL Offs(pOrigin,51.55,-38.36,-0.00),v40,z0,tcp\WObj:=Plywood;
    MoveL Offs(pOrigin,53.49,-41.44,-0.00),v40,z0,tcp\WObj:=Plywood;
    MoveL Offs(pOrigin,56.04,-44.21,-0.00),v40,z0,tcp\WObj:=Plywood;
    MoveL Offs(pOrigin,59.02,-46.15,-0.00),v40,z0,tcp\WObj:=Plywood;
    MoveL Offs(pOrigin,62.31,-47.18,-0.00),v40,z0,tcp\WObj:=Plywood;
    MoveL Offs(pOrigin,65.39,-47.39,-0.00),v40,z0,tcp\WObj:=Plywood;
    MoveL Offs(pOrigin,66.99,-46.65,-0.00),v40,z0,tcp\WObj:=Plywood;
    MoveL Offs(pOrigin,67.73,-45.76,-0.00),v40,z0,tcp\WObj:=Plywood;
    MoveL Offs(pOrigin,71.24,-44.10,-0.00),v40,z0,tcp\WObj:=Plywood;
    MoveL Offs(pOrigin,71.03,-43.89,-0.00),v40,z0,tcp\WObj:=Plywood;
    MoveL Offs(pOrigin,67.41,-44.53,-0.00),v40,z0,tcp\WObj:=Plywood;
    MoveL Offs(pOrigin,63.91,-44.53,-0.00),v40,z0,tcp\WObj:=Plywood;
    MoveL Offs(pOrigin,59.23,-43.39,-0.00),v40,z0,tcp\WObj:=Plywood;
    MoveL Offs(pOrigin,56.68,-41.87,-0.00),v40,z0,tcp\WObj:=Plywood;
    MoveL Offs(pOrigin,53.39,-37.94,-0.00),v40,z0,tcp\WObj:=Plywood;
    MoveL Offs(pOrigin,50.13,-34.96,-0.00),v40,fine,tcp\WObj:=Plywood;
    MoveL Offs(pOrigin,50.13,-34.96,-6.00),v60,z5,tcp\WObj:=Plywood;
    MoveL Offs(pOrigin,46.41,-36.10,-6.00),vTravel,z5,tcp\WObj:=Plywood;
    MoveL Offs(pOrigin,46.41,-36.10,-0.00),v60,z0,tcp\WObj:=Plywood;
    MoveL Offs(pOrigin,48.39,-39.00,-0.00),v40,z0,tcp\WObj:=Plywood;
    MoveL Offs(pOrigin,53.17,-43.46,-0.00),v40,z0,tcp\WObj:=Plywood;
    MoveL Offs(pOrigin,48.29,-39.64,-0.00),v40,z0,tcp\WObj:=Plywood;
    MoveL Offs(pOrigin,47.08,-37.94,-0.00),v40,z0,tcp\WObj:=Plywood;
    MoveL Offs(pOrigin,46.41,-36.10,-0.00),v40,fine,tcp\WObj:=Plywood;
    MoveL Offs(pOrigin,46.41,-36.10,-6.00),v60,z5,tcp\WObj:=Plywood;
    MoveL Offs(pOrigin,48.00,-41.09,-6.00),vTravel,z5,tcp\WObj:=Plywood;
    MoveL Offs(pOrigin,48.00,-41.09,-0.00),v60,z0,tcp\WObj:=Plywood;
    MoveL Offs(pOrigin,50.41,-43.25,-0.00),v40,z0,tcp\WObj:=Plywood;
    MoveL Offs(pOrigin,53.81,-45.62,-0.00),v40,z0,tcp\WObj:=Plywood;
    MoveL Offs(pOrigin,58.31,-47.68,-0.00),v40,z0,tcp\WObj:=Plywood;
    MoveL Offs(pOrigin,55.19,-46.79,-0.00),v40,z0,tcp\WObj:=Plywood;
    MoveL Offs(pOrigin,52.43,-45.30,-0.00),v40,z0,tcp\WObj:=Plywood;
    MoveL Offs(pOrigin,50.52,-43.89,-0.00),v40,z0,tcp\WObj:=Plywood;
    MoveL Offs(pOrigin,48.00,-41.09,-0.00),v40,fine,tcp\WObj:=Plywood;
    MoveL Offs(pOrigin,48.00,-41.09,-6.00),v60,z5,tcp\WObj:=Plywood;
    MoveL Offs(pOrigin,53.60,-52.03,-6.00),vTravel,z5,tcp\WObj:=Plywood;
    MoveL Offs(pOrigin,53.60,-52.03,-0.00),v60,z0,tcp\WObj:=Plywood;
    MoveL Offs(pOrigin,55.62,-55.26,-0.00),v40,z0,tcp\WObj:=Plywood;
    MoveL Offs(pOrigin,57.42,-57.06,-0.00),v40,z0,tcp\WObj:=Plywood;
    MoveL Offs(pOrigin,60.08,-58.59,-0.00),v40,z0,tcp\WObj:=Plywood;
    MoveL Offs(pOrigin,63.41,-59.72,-0.00),v40,z0,tcp\WObj:=Plywood;
    MoveL Offs(pOrigin,59.02,-58.48,-0.00),v40,z0,tcp\WObj:=Plywood;
    MoveL Offs(pOrigin,56.79,-57.06,-0.00),v40,z0,tcp\WObj:=Plywood;
    MoveL Offs(pOrigin,54.73,-54.51,-0.00),v40,z0,tcp\WObj:=Plywood;
    MoveL Offs(pOrigin,53.60,-52.03,-0.00),v40,fine,tcp\WObj:=Plywood;
    MoveL Offs(pOrigin,53.60,-52.03,-6.00),v60,z5,tcp\WObj:=Plywood;
    MoveL Offs(pOrigin,58.77,-59.90,-6.00),vTravel,z5,tcp\WObj:=Plywood;
    MoveL Offs(pOrigin,58.77,-59.90,-0.00),v60,z0,tcp\WObj:=Plywood;
    MoveL Offs(pOrigin,63.27,-62.23,-0.00),v40,z0,tcp\WObj:=Plywood;
    MoveL Offs(pOrigin,65.29,-63.65,-0.00),v40,z0,tcp\WObj:=Plywood;
    MoveL Offs(pOrigin,65.85,-64.54,-0.00),v40,z0,tcp\WObj:=Plywood;
    MoveL Offs(pOrigin,58.77,-59.90,-0.00),v40,fine,tcp\WObj:=Plywood;
    MoveL Offs(pOrigin,58.77,-59.90,-6.00),v60,z5,tcp\WObj:=Plywood;
    MoveL Offs(pOrigin,69.40,-60.78,-6.00),vTravel,z5,tcp\WObj:=Plywood;
    MoveL Offs(pOrigin,69.40,-60.78,-0.00),v60,z0,tcp\WObj:=Plywood;
    MoveL Offs(pOrigin,74.32,-62.06,-0.00),v40,z0,tcp\WObj:=Plywood;
    MoveL Offs(pOrigin,78.75,-62.34,-0.00),v40,z0,tcp\WObj:=Plywood;
    MoveL Offs(pOrigin,77.61,-62.59,-0.00),v40,z0,tcp\WObj:=Plywood;
    MoveL Offs(pOrigin,74.32,-62.38,-0.00),v40,z0,tcp\WObj:=Plywood;
    MoveL Offs(pOrigin,69.40,-60.78,-0.00),v40,fine,tcp\WObj:=Plywood;
    MoveL Offs(pOrigin,69.40,-60.78,-6.00),v60,z5,tcp\WObj:=Plywood;
    MoveL Offs(pOrigin,66.63,-50.58,-6.00),vTravel,z5,tcp\WObj:=Plywood;
    MoveL Offs(pOrigin,66.63,-50.58,-0.00),v60,z0,tcp\WObj:=Plywood;
    MoveL Offs(pOrigin,69.64,-49.87,-0.00),v40,z0,tcp\WObj:=Plywood;
    MoveL Offs(pOrigin,73.15,-48.14,-0.00),v40,z0,tcp\WObj:=Plywood;
    MoveL Offs(pOrigin,76.12,-45.59,-0.00),v40,z0,tcp\WObj:=Plywood;
    MoveL Offs(pOrigin,78.57,-42.61,-0.00),v40,z0,tcp\WObj:=Plywood;
    MoveL Offs(pOrigin,76.34,-45.91,-0.00),v40,z0,tcp\WObj:=Plywood;
    MoveL Offs(pOrigin,74.21,-47.82,-0.00),v40,z0,tcp\WObj:=Plywood;
    MoveL Offs(pOrigin,70.92,-49.66,-0.00),v40,z0,tcp\WObj:=Plywood;
    MoveL Offs(pOrigin,66.63,-50.58,-0.00),v40,fine,tcp\WObj:=Plywood;
    MoveL Offs(pOrigin,66.63,-50.58,-6.00),v60,z5,tcp\WObj:=Plywood;
    MoveL Offs(pOrigin,67.94,-46.30,-6.00),vTravel,z5,tcp\WObj:=Plywood;
    MoveL Offs(pOrigin,67.94,-46.30,-0.00),v60,z0,tcp\WObj:=Plywood;
    MoveL Offs(pOrigin,69.43,-45.30,-0.00),v40,z0,tcp\WObj:=Plywood;
    MoveL Offs(pOrigin,67.94,-46.30,-0.00),v40,fine,tcp\WObj:=Plywood;
    MoveL Offs(pOrigin,67.94,-46.30,-6.00),v60,z5,tcp\WObj:=Plywood;
    MoveL Offs(pOrigin,72.16,-47.15,-6.00),vTravel,z5,tcp\WObj:=Plywood;
    MoveL Offs(pOrigin,72.16,-47.15,-0.00),v60,z0,tcp\WObj:=Plywood;
    MoveL Offs(pOrigin,76.59,-42.75,-0.00),v40,z0,tcp\WObj:=Plywood;
    MoveL Offs(pOrigin,72.16,-47.15,-0.00),v40,fine,tcp\WObj:=Plywood;
    MoveL Offs(pOrigin,72.16,-47.15,-6.00),v60,z5,tcp\WObj:=Plywood;
    MoveL Offs(pOrigin,76.12,-39.42,-6.00),vTravel,z5,tcp\WObj:=Plywood;
    MoveL Offs(pOrigin,76.12,-39.42,-0.00),v60,z0,tcp\WObj:=Plywood;
    MoveL Offs(pOrigin,79.74,-39.32,-0.00),v40,z0,tcp\WObj:=Plywood;
    MoveL Offs(pOrigin,82.39,-38.50,-0.00),v40,z0,tcp\WObj:=Plywood;
    MoveL Offs(pOrigin,83.67,-37.72,-0.00),v40,z0,tcp\WObj:=Plywood;
    MoveL Offs(pOrigin,83.67,-37.41,-0.00),v40,z0,tcp\WObj:=Plywood;
    MoveL Offs(pOrigin,83.03,-37.19,-0.00),v40,z0,tcp\WObj:=Plywood;
    MoveL Offs(pOrigin,80.69,-38.26,-0.00),v40,z0,tcp\WObj:=Plywood;
    MoveL Offs(pOrigin,78.78,-38.47,-0.00),v40,z0,tcp\WObj:=Plywood;
    MoveL Offs(pOrigin,75.59,-37.65,-0.00),v40,z0,tcp\WObj:=Plywood;
    MoveL Offs(pOrigin,71.13,-34.75,-0.00),v40,z0,tcp\WObj:=Plywood;
    MoveL Offs(pOrigin,69.32,-32.84,-0.00),v40,z0,tcp\WObj:=Plywood;
    MoveL Offs(pOrigin,68.33,-31.14,-0.00),v40,z0,tcp\WObj:=Plywood;
    MoveL Offs(pOrigin,67.94,-29.65,-0.00),v40,z0,tcp\WObj:=Plywood;
    MoveL Offs(pOrigin,68.16,-27.31,-0.00),v40,z0,tcp\WObj:=Plywood;
    MoveL Offs(pOrigin,68.76,-25.83,-0.00),v40,z0,tcp\WObj:=Plywood;
    MoveL Offs(pOrigin,70.39,-23.59,-0.00),v40,z0,tcp\WObj:=Plywood;
    MoveL Offs(pOrigin,72.62,-21.96,-0.00),v40,z0,tcp\WObj:=Plywood;
    MoveL Offs(pOrigin,73.68,-21.68,-0.00),v40,z0,tcp\WObj:=Plywood;
    MoveL Offs(pOrigin,76.34,-21.86,-0.00),v40,z0,tcp\WObj:=Plywood;
    MoveL Offs(pOrigin,76.66,-21.68,-0.00),v40,z0,tcp\WObj:=Plywood;
    MoveL Offs(pOrigin,76.55,-21.40,-0.00),v40,z0,tcp\WObj:=Plywood;
    MoveL Offs(pOrigin,74.43,-20.94,-0.00),v40,z0,tcp\WObj:=Plywood;
    MoveL Offs(pOrigin,72.19,-21.22,-0.00),v40,z0,tcp\WObj:=Plywood;
    MoveL Offs(pOrigin,69.96,-22.85,-0.00),v40,z0,tcp\WObj:=Plywood;
    MoveL Offs(pOrigin,68.55,-25.01,-0.00),v40,z0,tcp\WObj:=Plywood;
    MoveL Offs(pOrigin,69.64,-22.74,-0.00),v40,z0,tcp\WObj:=Plywood;
    MoveL Offs(pOrigin,71.10,-21.26,-0.00),v40,z0,tcp\WObj:=Plywood;
    MoveL Offs(pOrigin,68.58,-21.58,-0.00),v40,z0,tcp\WObj:=Plywood;
    MoveL Offs(pOrigin,65.71,-22.85,-0.00),v40,z0,tcp\WObj:=Plywood;
    MoveL Offs(pOrigin,64.08,-24.59,-0.00),v40,z0,tcp\WObj:=Plywood;
    MoveL Offs(pOrigin,65.25,-23.06,-0.00),v40,z0,tcp\WObj:=Plywood;
    MoveL Offs(pOrigin,65.07,-22.89,-0.00),v40,z0,tcp\WObj:=Plywood;
  ENDPROC

  PROC DrawPart5()
    MoveL Offs(pOrigin,63.02,-25.08,-0.00),v40,z0,tcp\WObj:=Plywood;
    MoveL Offs(pOrigin,62.42,-27.10,-0.00),v40,z0,tcp\WObj:=Plywood;
    MoveL Offs(pOrigin,62.42,-28.48,-0.00),v40,z0,tcp\WObj:=Plywood;
    MoveL Offs(pOrigin,63.02,-30.82,-0.00),v40,z0,tcp\WObj:=Plywood;
    MoveL Offs(pOrigin,65.07,-34.22,-0.00),v40,z0,tcp\WObj:=Plywood;
    MoveL Offs(pOrigin,67.41,-36.17,-0.00),v40,z0,tcp\WObj:=Plywood;
    MoveL Offs(pOrigin,71.34,-38.08,-0.00),v40,z0,tcp\WObj:=Plywood;
    MoveL Offs(pOrigin,76.12,-39.42,-0.00),v40,fine,tcp\WObj:=Plywood;
    MoveL Offs(pOrigin,76.12,-39.42,-6.00),v60,z5,tcp\WObj:=Plywood;
    MoveL Offs(pOrigin,76.73,-37.19,-6.00),vTravel,z5,tcp\WObj:=Plywood;
    MoveL Offs(pOrigin,76.73,-37.19,-0.00),v60,z0,tcp\WObj:=Plywood;
    MoveL Offs(pOrigin,78.78,-37.83,-0.00),v40,z0,tcp\WObj:=Plywood;
    MoveL Offs(pOrigin,80.27,-37.72,-0.00),v40,z0,tcp\WObj:=Plywood;
    MoveL Offs(pOrigin,81.05,-37.30,-0.00),v40,z0,tcp\WObj:=Plywood;
    MoveL Offs(pOrigin,78.99,-37.51,-0.00),v40,z0,tcp\WObj:=Plywood;
    MoveL Offs(pOrigin,76.73,-37.19,-0.00),v40,z0,tcp\WObj:=Plywood;
    MoveL Offs(pOrigin,76.66,-37.16,-0.00),v40,z0,tcp\WObj:=Plywood;
    MoveL Offs(pOrigin,72.34,-33.79,-0.00),v40,z0,tcp\WObj:=Plywood;
    MoveL Offs(pOrigin,73.89,-35.60,-0.00),v40,z0,tcp\WObj:=Plywood;
    MoveL Offs(pOrigin,76.66,-37.16,-0.00),v40,z0,tcp\WObj:=Plywood;
    MoveL Offs(pOrigin,76.87,-36.70,-0.00),v40,z0,tcp\WObj:=Plywood;
    MoveL Offs(pOrigin,78.36,-37.05,-0.00),v40,z0,tcp\WObj:=Plywood;
    MoveL Offs(pOrigin,75.91,-35.71,-0.00),v40,z0,tcp\WObj:=Plywood;
    MoveL Offs(pOrigin,73.89,-33.79,-0.00),v40,z0,tcp\WObj:=Plywood;
    MoveL Offs(pOrigin,71.13,-29.05,-0.00),v40,z0,tcp\WObj:=Plywood;
    MoveL Offs(pOrigin,72.37,-32.20,-0.00),v40,z0,tcp\WObj:=Plywood;
    MoveL Offs(pOrigin,74.96,-35.17,-0.00),v40,z0,tcp\WObj:=Plywood;
    MoveL Offs(pOrigin,75.06,-35.67,-0.00),v40,z0,tcp\WObj:=Plywood;
    MoveL Offs(pOrigin,76.87,-36.70,-0.00),v40,fine,tcp\WObj:=Plywood;
    MoveL Offs(pOrigin,76.87,-36.70,-6.00),v60,z5,tcp\WObj:=Plywood;
    MoveL Offs(pOrigin,76.12,-35.07,-6.00),vTravel,z5,tcp\WObj:=Plywood;
    MoveL Offs(pOrigin,76.12,-35.07,-0.00),v60,z0,tcp\WObj:=Plywood;
    MoveL Offs(pOrigin,79.10,-36.45,-0.00),v40,z0,tcp\WObj:=Plywood;
    MoveL Offs(pOrigin,83.24,-36.63,-0.00),v40,z0,tcp\WObj:=Plywood;
    MoveL Offs(pOrigin,81.83,-35.25,-0.00),v40,z0,tcp\WObj:=Plywood;
    MoveL Offs(pOrigin,82.61,-35.56,-0.00),v40,z0,tcp\WObj:=Plywood;
    MoveL Offs(pOrigin,87.71,-39.96,-0.00),v40,z0,tcp\WObj:=Plywood;
    MoveL Offs(pOrigin,89.72,-41.02,-0.00),v40,z0,tcp\WObj:=Plywood;
    MoveL Offs(pOrigin,91.21,-41.02,-0.00),v40,z0,tcp\WObj:=Plywood;
    MoveL Offs(pOrigin,93.97,-40.20,-0.00),v40,z0,tcp\WObj:=Plywood;
    MoveL Offs(pOrigin,102.05,-36.80,-0.00),v40,z0,tcp\WObj:=Plywood;
    MoveL Offs(pOrigin,106.72,-33.26,-0.00),v40,z0,tcp\WObj:=Plywood;
    MoveL Offs(pOrigin,108.00,-31.99,-0.00),v40,z0,tcp\WObj:=Plywood;
    MoveL Offs(pOrigin,108.46,-30.82,-0.00),v40,z0,tcp\WObj:=Plywood;
    MoveL Offs(pOrigin,107.79,-29.33,-0.00),v40,z0,tcp\WObj:=Plywood;
    MoveL Offs(pOrigin,106.41,-28.91,-0.00),v40,z0,tcp\WObj:=Plywood;
    MoveL Offs(pOrigin,100.78,-31.81,-0.00),v40,z0,tcp\WObj:=Plywood;
    MoveL Offs(pOrigin,91.81,-34.82,-0.00),v40,z0,tcp\WObj:=Plywood;
    MoveL Offs(pOrigin,92.81,-33.86,-0.00),v40,z0,tcp\WObj:=Plywood;
    MoveL Offs(pOrigin,99.29,-31.81,-0.00),v40,z0,tcp\WObj:=Plywood;
    MoveL Offs(pOrigin,102.58,-30.32,-0.00),v40,z0,tcp\WObj:=Plywood;
    MoveL Offs(pOrigin,106.41,-27.95,-0.00),v40,z0,tcp\WObj:=Plywood;
    MoveL Offs(pOrigin,107.57,-26.46,-0.00),v40,z0,tcp\WObj:=Plywood;
    MoveL Offs(pOrigin,107.50,-25.29,-0.00),v40,z0,tcp\WObj:=Plywood;
    MoveL Offs(pOrigin,106.83,-24.44,-0.00),v40,z0,tcp\WObj:=Plywood;
    MoveL Offs(pOrigin,105.13,-24.02,-0.00),v40,z0,tcp\WObj:=Plywood;
    MoveL Offs(pOrigin,97.16,-26.14,-0.00),v40,z0,tcp\WObj:=Plywood;
    MoveL Offs(pOrigin,90.79,-28.59,-0.00),v40,z0,tcp\WObj:=Plywood;
    MoveL Offs(pOrigin,94.40,-26.36,-0.00),v40,z0,tcp\WObj:=Plywood;
    MoveL Offs(pOrigin,93.87,-25.29,-0.00),v40,z0,tcp\WObj:=Plywood;
    MoveL Offs(pOrigin,92.45,-24.23,-0.00),v40,z0,tcp\WObj:=Plywood;
    MoveL Offs(pOrigin,92.38,-22.35,-0.00),v40,z0,tcp\WObj:=Plywood;
    MoveL Offs(pOrigin,89.62,-23.10,-0.00),v40,z0,tcp\WObj:=Plywood;
    MoveL Offs(pOrigin,93.87,-21.15,-0.00),v40,z0,tcp\WObj:=Plywood;
    MoveL Offs(pOrigin,97.38,-20.41,-0.00),v40,z0,tcp\WObj:=Plywood;
    MoveL Offs(pOrigin,99.89,-20.30,-0.00),v40,z0,tcp\WObj:=Plywood;
    MoveL Offs(pOrigin,98.86,-19.41,-0.00),v40,z0,tcp\WObj:=Plywood;
    MoveL Offs(pOrigin,95.99,-18.71,-0.00),v40,z0,tcp\WObj:=Plywood;
    MoveL Offs(pOrigin,93.44,-18.60,-0.00),v40,z0,tcp\WObj:=Plywood;
    MoveL Offs(pOrigin,88.88,-19.02,-0.00),v40,z0,tcp\WObj:=Plywood;
    MoveL Offs(pOrigin,86.32,-18.71,-0.00),v40,z0,tcp\WObj:=Plywood;
    MoveL Offs(pOrigin,81.86,-19.41,-0.00),v40,z0,tcp\WObj:=Plywood;
    MoveL Offs(pOrigin,76.66,-22.46,-0.00),v40,z0,tcp\WObj:=Plywood;
    MoveL Offs(pOrigin,73.04,-23.81,-0.00),v40,z0,tcp\WObj:=Plywood;
    MoveL Offs(pOrigin,71.84,-25.40,-0.00),v40,z0,tcp\WObj:=Plywood;
    MoveL Offs(pOrigin,71.56,-27.42,-0.00),v40,z0,tcp\WObj:=Plywood;
    MoveL Offs(pOrigin,72.90,-31.24,-0.00),v40,z0,tcp\WObj:=Plywood;
    MoveL Offs(pOrigin,74.00,-32.94,-0.00),v40,z0,tcp\WObj:=Plywood;
    MoveL Offs(pOrigin,76.12,-35.07,-0.00),v40,fine,tcp\WObj:=Plywood;
    MoveL Offs(pOrigin,76.12,-35.07,-6.00),v60,z5,tcp\WObj:=Plywood;
    MoveL Offs(pOrigin,74.96,-35.56,-6.00),vTravel,z5,tcp\WObj:=Plywood;
    MoveL Offs(pOrigin,74.96,-35.56,-0.00),v60,z0,tcp\WObj:=Plywood;
    MoveL Offs(pOrigin,74.32,-35.00,-0.00),v40,z0,tcp\WObj:=Plywood;
    MoveL Offs(pOrigin,74.96,-35.56,-0.00),v40,fine,tcp\WObj:=Plywood;
    MoveL Offs(pOrigin,74.96,-35.56,-6.00),v60,z5,tcp\WObj:=Plywood;
    MoveL Offs(pOrigin,73.89,-34.82,-6.00),vTravel,z5,tcp\WObj:=Plywood;
    MoveL Offs(pOrigin,73.89,-34.82,-0.00),v60,z0,tcp\WObj:=Plywood;
    MoveL Offs(pOrigin,72.05,-32.41,-0.00),v40,z0,tcp\WObj:=Plywood;
    MoveL Offs(pOrigin,70.39,-29.15,-0.00),v40,z0,tcp\WObj:=Plywood;
    MoveL Offs(pOrigin,70.78,-30.92,-0.00),v40,z0,tcp\WObj:=Plywood;
    MoveL Offs(pOrigin,72.72,-33.90,-0.00),v40,z0,tcp\WObj:=Plywood;
    MoveL Offs(pOrigin,73.89,-34.82,-0.00),v40,fine,tcp\WObj:=Plywood;
    MoveL Offs(pOrigin,73.89,-34.82,-6.00),v60,z5,tcp\WObj:=Plywood;
    MoveL Offs(pOrigin,71.88,-34.47,-6.00),vTravel,z5,tcp\WObj:=Plywood;
    MoveL Offs(pOrigin,71.88,-34.47,-0.00),v60,z0,tcp\WObj:=Plywood;
    MoveL Offs(pOrigin,69.82,-31.03,-0.00),v40,z0,tcp\WObj:=Plywood;
    MoveL Offs(pOrigin,68.79,-28.02,-0.00),v40,z0,tcp\WObj:=Plywood;
    MoveL Offs(pOrigin,68.58,-29.76,-0.00),v40,z0,tcp\WObj:=Plywood;
    MoveL Offs(pOrigin,68.97,-31.03,-0.00),v40,z0,tcp\WObj:=Plywood;
    MoveL Offs(pOrigin,70.07,-32.73,-0.00),v40,z0,tcp\WObj:=Plywood;
    MoveL Offs(pOrigin,71.88,-34.47,-0.00),v40,fine,tcp\WObj:=Plywood;
    MoveL Offs(pOrigin,71.88,-34.47,-6.00),v60,z5,tcp\WObj:=Plywood;
    MoveL Offs(pOrigin,71.45,-32.73,-6.00),vTravel,z5,tcp\WObj:=Plywood;
    MoveL Offs(pOrigin,71.45,-32.73,-0.00),v60,z0,tcp\WObj:=Plywood;
    MoveL Offs(pOrigin,71.24,-32.20,-0.00),v40,z0,tcp\WObj:=Plywood;
    MoveL Offs(pOrigin,71.45,-32.73,-0.00),v40,fine,tcp\WObj:=Plywood;
    MoveL Offs(pOrigin,71.45,-32.73,-6.00),v60,z5,tcp\WObj:=Plywood;
    MoveL Offs(pOrigin,70.81,-31.60,-6.00),vTravel,z5,tcp\WObj:=Plywood;
    MoveL Offs(pOrigin,70.81,-31.60,-0.00),v60,z0,tcp\WObj:=Plywood;
    MoveL Offs(pOrigin,70.60,-31.00,-0.00),v40,z0,tcp\WObj:=Plywood;
    MoveL Offs(pOrigin,70.81,-31.60,-0.00),v40,fine,tcp\WObj:=Plywood;
    MoveL Offs(pOrigin,70.81,-31.60,-6.00),v60,z5,tcp\WObj:=Plywood;
    MoveL Offs(pOrigin,70.28,-28.80,-6.00),vTravel,z5,tcp\WObj:=Plywood;
    MoveL Offs(pOrigin,70.28,-28.80,-0.00),v60,z0,tcp\WObj:=Plywood;
    MoveL Offs(pOrigin,70.49,-28.48,-0.00),v40,z0,tcp\WObj:=Plywood;
    MoveL Offs(pOrigin,70.18,-28.27,-0.00),v40,z0,tcp\WObj:=Plywood;
    MoveL Offs(pOrigin,70.28,-28.80,-0.00),v40,z0,tcp\WObj:=Plywood;
    MoveL Offs(pOrigin,70.49,-28.48,-0.00),v40,z0,tcp\WObj:=Plywood;
    MoveL Offs(pOrigin,70.07,-28.38,-0.00),v40,z0,tcp\WObj:=Plywood;
    MoveL Offs(pOrigin,70.28,-28.80,-0.00),v40,z0,tcp\WObj:=Plywood;
  ENDPROC

  PROC DrawPart6()
    MoveL Offs(pOrigin,70.81,-28.27,-0.00),v40,z0,tcp\WObj:=Plywood;
    MoveL Offs(pOrigin,71.03,-28.69,-0.00),v40,z0,tcp\WObj:=Plywood;
    MoveL Offs(pOrigin,71.24,-28.38,-0.00),v40,z0,tcp\WObj:=Plywood;
    MoveL Offs(pOrigin,70.92,-28.16,-0.00),v40,z0,tcp\WObj:=Plywood;
    MoveL Offs(pOrigin,71.03,-28.69,-0.00),v40,z0,tcp\WObj:=Plywood;
    MoveL Offs(pOrigin,71.24,-28.38,-0.00),v40,z0,tcp\WObj:=Plywood;
    MoveL Offs(pOrigin,70.81,-28.27,-0.00),v40,z0,tcp\WObj:=Plywood;
    MoveL Offs(pOrigin,70.81,-27.70,-0.00),v40,z0,tcp\WObj:=Plywood;
    MoveL Offs(pOrigin,71.03,-25.58,-0.00),v40,z0,tcp\WObj:=Plywood;
    MoveL Offs(pOrigin,70.60,-26.78,-0.00),v40,z0,tcp\WObj:=Plywood;
    MoveL Offs(pOrigin,70.81,-27.70,-0.00),v40,z0,tcp\WObj:=Plywood;
    MoveL Offs(pOrigin,70.07,-27.81,-0.00),v40,z0,tcp\WObj:=Plywood;
    MoveL Offs(pOrigin,70.88,-25.19,-0.00),v40,z0,tcp\WObj:=Plywood;
    MoveL Offs(pOrigin,71.88,-23.70,-0.00),v40,z0,tcp\WObj:=Plywood;
    MoveL Offs(pOrigin,74.64,-22.35,-0.00),v40,z0,tcp\WObj:=Plywood;
    MoveL Offs(pOrigin,72.94,-22.60,-0.00),v40,z0,tcp\WObj:=Plywood;
    MoveL Offs(pOrigin,71.24,-23.81,-0.00),v40,z0,tcp\WObj:=Plywood;
    MoveL Offs(pOrigin,70.28,-25.51,-0.00),v40,z0,tcp\WObj:=Plywood;
    MoveL Offs(pOrigin,70.07,-27.81,-0.00),v40,z0,tcp\WObj:=Plywood;
    MoveL Offs(pOrigin,69.64,-27.63,-0.00),v40,z0,tcp\WObj:=Plywood;
    MoveL Offs(pOrigin,69.64,-25.79,-0.00),v40,z0,tcp\WObj:=Plywood;
    MoveL Offs(pOrigin,69.01,-26.99,-0.00),v40,z0,tcp\WObj:=Plywood;
    MoveL Offs(pOrigin,69.32,-27.84,-0.00),v40,z0,tcp\WObj:=Plywood;
    MoveL Offs(pOrigin,69.64,-27.63,-0.00),v40,fine,tcp\WObj:=Plywood;
    MoveL Offs(pOrigin,69.64,-27.63,-6.00),v60,z5,tcp\WObj:=Plywood;
    MoveL Offs(pOrigin,61.99,-28.06,-6.00),vTravel,z5,tcp\WObj:=Plywood;
    MoveL Offs(pOrigin,61.99,-28.06,-0.00),v60,z0,tcp\WObj:=Plywood;
    MoveL Offs(pOrigin,62.10,-25.19,-0.00),v40,z0,tcp\WObj:=Plywood;
    MoveL Offs(pOrigin,63.34,-22.85,-0.00),v40,z0,tcp\WObj:=Plywood;
    MoveL Offs(pOrigin,62.63,-22.64,-0.00),v40,z0,tcp\WObj:=Plywood;
    MoveL Offs(pOrigin,61.78,-23.27,-0.00),v40,z0,tcp\WObj:=Plywood;
    MoveL Offs(pOrigin,60.79,-24.87,-0.00),v40,z0,tcp\WObj:=Plywood;
    MoveL Offs(pOrigin,60.51,-27.10,-0.00),v40,z0,tcp\WObj:=Plywood;
    MoveL Offs(pOrigin,61.96,-30.61,-0.00),v40,z0,tcp\WObj:=Plywood;
    MoveL Offs(pOrigin,63.69,-32.87,-0.00),v40,z0,tcp\WObj:=Plywood;
    MoveL Offs(pOrigin,61.99,-28.06,-0.00),v40,fine,tcp\WObj:=Plywood;
    MoveL Offs(pOrigin,61.99,-28.06,-6.00),v60,z5,tcp\WObj:=Plywood;
    MoveL Offs(pOrigin,60.75,-29.23,-6.00),vTravel,z5,tcp\WObj:=Plywood;
    MoveL Offs(pOrigin,60.75,-29.23,-0.00),v60,z0,tcp\WObj:=Plywood;
    MoveL Offs(pOrigin,60.93,-30.50,-0.00),v40,z0,tcp\WObj:=Plywood;
    MoveL Offs(pOrigin,61.78,-32.52,-0.00),v40,z0,tcp\WObj:=Plywood;
    MoveL Offs(pOrigin,63.38,-34.01,-0.00),v40,z0,tcp\WObj:=Plywood;
    MoveL Offs(pOrigin,65.25,-35.07,-0.00),v40,z0,tcp\WObj:=Plywood;
    MoveL Offs(pOrigin,62.84,-32.31,-0.00),v40,z0,tcp\WObj:=Plywood;
    MoveL Offs(pOrigin,60.75,-29.23,-0.00),v40,fine,tcp\WObj:=Plywood;
    MoveL Offs(pOrigin,60.75,-29.23,-6.00),v60,z5,tcp\WObj:=Plywood;
    MoveL Offs(pOrigin,57.53,-24.51,-6.00),vTravel,z5,tcp\WObj:=Plywood;
    MoveL Offs(pOrigin,57.53,-24.51,-0.00),v60,z0,tcp\WObj:=Plywood;
    MoveL Offs(pOrigin,58.42,-23.70,-0.00),v40,z0,tcp\WObj:=Plywood;
    MoveL Offs(pOrigin,58.59,-22.25,-0.00),v40,z0,tcp\WObj:=Plywood;
    MoveL Offs(pOrigin,57.96,-22.32,-0.00),v40,z0,tcp\WObj:=Plywood;
    MoveL Offs(pOrigin,57.50,-23.06,-0.00),v40,z0,tcp\WObj:=Plywood;
    MoveL Offs(pOrigin,57.53,-24.51,-0.00),v40,z0,tcp\WObj:=Plywood;
    MoveL Offs(pOrigin,57.04,-24.02,-0.00),v40,z0,tcp\WObj:=Plywood;
    MoveL Offs(pOrigin,57.32,-22.14,-0.00),v40,z0,tcp\WObj:=Plywood;
    MoveL Offs(pOrigin,56.68,-22.64,-0.00),v40,z0,tcp\WObj:=Plywood;
    MoveL Offs(pOrigin,56.26,-23.59,-0.00),v40,z0,tcp\WObj:=Plywood;
    MoveL Offs(pOrigin,56.58,-24.66,-0.00),v40,z0,tcp\WObj:=Plywood;
    MoveL Offs(pOrigin,57.04,-24.02,-0.00),v40,z0,tcp\WObj:=Plywood;
    MoveL Offs(pOrigin,56.04,-24.55,-0.00),v40,z0,tcp\WObj:=Plywood;
    MoveL Offs(pOrigin,56.04,-23.10,-0.00),v40,z0,tcp\WObj:=Plywood;
    MoveL Offs(pOrigin,55.41,-24.34,-0.00),v40,z0,tcp\WObj:=Plywood;
    MoveL Offs(pOrigin,55.72,-24.87,-0.00),v40,z0,tcp\WObj:=Plywood;
    MoveL Offs(pOrigin,56.04,-24.55,-0.00),v40,fine,tcp\WObj:=Plywood;
    MoveL Offs(pOrigin,56.04,-24.55,-6.00),v60,z5,tcp\WObj:=Plywood;
    MoveL Offs(pOrigin,60.86,-23.38,-6.00),vTravel,z5,tcp\WObj:=Plywood;
    MoveL Offs(pOrigin,60.86,-23.38,-0.00),v60,z0,tcp\WObj:=Plywood;
    MoveL Offs(pOrigin,61.36,-22.57,-0.00),v40,z0,tcp\WObj:=Plywood;
    MoveL Offs(pOrigin,61.00,-22.74,-0.00),v40,z0,tcp\WObj:=Plywood;
    MoveL Offs(pOrigin,60.86,-23.38,-0.00),v40,fine,tcp\WObj:=Plywood;
    MoveL Offs(pOrigin,60.86,-23.38,-6.00),v60,z5,tcp\WObj:=Plywood;
    MoveL Offs(pOrigin,81.83,-34.68,-6.00),vTravel,z5,tcp\WObj:=Plywood;
    MoveL Offs(pOrigin,81.83,-34.68,-0.00),v60,z0,tcp\WObj:=Plywood;
    MoveL Offs(pOrigin,80.52,-32.80,-0.00),v40,z0,tcp\WObj:=Plywood;
    MoveL Offs(pOrigin,81.83,-34.68,-0.00),v40,fine,tcp\WObj:=Plywood;
    MoveL Offs(pOrigin,81.83,-34.68,-6.00),v60,z5,tcp\WObj:=Plywood;
    MoveL Offs(pOrigin,84.20,-39.60,-6.00),vTravel,z5,tcp\WObj:=Plywood;
    MoveL Offs(pOrigin,84.20,-39.60,-0.00),v60,z0,tcp\WObj:=Plywood;
    MoveL Offs(pOrigin,79.84,-41.23,-0.00),v40,z0,tcp\WObj:=Plywood;
    MoveL Offs(pOrigin,80.69,-44.21,-0.00),v40,z0,tcp\WObj:=Plywood;
    MoveL Offs(pOrigin,81.12,-48.85,-0.00),v40,z0,tcp\WObj:=Plywood;
    MoveL Offs(pOrigin,84.20,-39.60,-0.00),v40,z0,tcp\WObj:=Plywood;
    MoveL Offs(pOrigin,85.16,-39.21,-0.00),v40,z0,tcp\WObj:=Plywood;
    MoveL Offs(pOrigin,84.16,-41.12,-0.00),v40,z0,tcp\WObj:=Plywood;
    MoveL Offs(pOrigin,82.71,-44.95,-0.00),v40,z0,tcp\WObj:=Plywood;
    MoveL Offs(pOrigin,81.65,-49.41,-0.00),v40,z0,tcp\WObj:=Plywood;
    MoveL Offs(pOrigin,82.07,-50.62,-0.00),v40,z0,tcp\WObj:=Plywood;
    MoveL Offs(pOrigin,82.78,-48.99,-0.00),v40,z0,tcp\WObj:=Plywood;
    MoveL Offs(pOrigin,83.78,-47.71,-0.00),v40,z0,tcp\WObj:=Plywood;
    MoveL Offs(pOrigin,90.22,-41.87,-0.00),v40,z0,tcp\WObj:=Plywood;
    MoveL Offs(pOrigin,88.34,-41.20,-0.00),v40,z0,tcp\WObj:=Plywood;
    MoveL Offs(pOrigin,85.69,-38.93,-0.00),v40,z0,tcp\WObj:=Plywood;
    MoveL Offs(pOrigin,85.16,-39.21,-0.00),v40,fine,tcp\WObj:=Plywood;
    MoveL Offs(pOrigin,85.16,-39.21,-6.00),v60,z5,tcp\WObj:=Plywood;
    MoveL Offs(pOrigin,91.32,-41.87,-6.00),vTravel,z5,tcp\WObj:=Plywood;
    MoveL Offs(pOrigin,91.32,-41.87,-0.00),v60,z0,tcp\WObj:=Plywood;
    MoveL Offs(pOrigin,84.94,-47.50,-0.00),v40,z0,tcp\WObj:=Plywood;
    MoveL Offs(pOrigin,83.67,-49.31,-0.00),v40,z0,tcp\WObj:=Plywood;
    MoveL Offs(pOrigin,84.91,-50.26,-0.00),v40,z0,tcp\WObj:=Plywood;
    MoveL Offs(pOrigin,94.29,-42.05,-0.00),v40,z0,tcp\WObj:=Plywood;
    MoveL Offs(pOrigin,94.19,-41.44,-0.00),v40,z0,tcp\WObj:=Plywood;
    MoveL Offs(pOrigin,93.66,-41.02,-0.00),v40,z0,tcp\WObj:=Plywood;
    MoveL Offs(pOrigin,93.23,-41.16,-0.00),v40,z0,tcp\WObj:=Plywood;
    MoveL Offs(pOrigin,93.30,-41.51,-0.00),v40,z0,tcp\WObj:=Plywood;
    MoveL Offs(pOrigin,84.20,-49.38,-0.00),v40,z0,tcp\WObj:=Plywood;
    MoveL Offs(pOrigin,93.09,-41.34,-0.00),v40,z0,tcp\WObj:=Plywood;
    MoveL Offs(pOrigin,91.32,-41.87,-0.00),v40,fine,tcp\WObj:=Plywood;
    MoveL Offs(pOrigin,91.32,-41.87,-6.00),v60,z5,tcp\WObj:=Plywood;
    MoveL Offs(pOrigin,93.97,-42.72,-6.00),vTravel,z5,tcp\WObj:=Plywood;
    MoveL Offs(pOrigin,93.97,-42.72,-0.00),v60,z0,tcp\WObj:=Plywood;
    MoveL Offs(pOrigin,94.08,-43.00,-0.00),v40,z0,tcp\WObj:=Plywood;
    MoveL Offs(pOrigin,94.65,-42.51,-0.00),v40,z0,tcp\WObj:=Plywood;
    MoveL Offs(pOrigin,94.51,-42.08,-0.00),v40,z0,tcp\WObj:=Plywood;
    MoveL Offs(pOrigin,93.97,-42.72,-0.00),v40,z0,tcp\WObj:=Plywood;
    MoveL Offs(pOrigin,93.87,-43.04,-0.00),v40,z0,tcp\WObj:=Plywood;
    MoveL Offs(pOrigin,84.98,-50.37,-0.00),v40,z0,tcp\WObj:=Plywood;
    MoveL Offs(pOrigin,85.47,-50.40,-0.00),v40,z0,tcp\WObj:=Plywood;
    MoveL Offs(pOrigin,93.23,-44.10,-0.00),v40,z0,tcp\WObj:=Plywood;
    MoveL Offs(pOrigin,93.94,-43.36,-0.00),v40,z0,tcp\WObj:=Plywood;
    MoveL Offs(pOrigin,93.87,-43.04,-0.00),v40,z0,tcp\WObj:=Plywood;
  ENDPROC

  PROC DrawPart7()
    MoveL Offs(pOrigin,94.82,-43.46,-0.00),v40,z0,tcp\WObj:=Plywood;
    MoveL Offs(pOrigin,86.64,-50.47,-0.00),v40,z0,tcp\WObj:=Plywood;
    MoveL Offs(pOrigin,95.39,-59.65,-0.00),v40,z0,tcp\WObj:=Plywood;
    MoveL Offs(pOrigin,86.54,-50.79,-0.00),v40,z0,tcp\WObj:=Plywood;
    MoveL Offs(pOrigin,84.20,-51.43,-0.00),v40,z0,tcp\WObj:=Plywood;
    MoveL Offs(pOrigin,83.46,-51.25,-0.00),v40,z0,tcp\WObj:=Plywood;
    MoveL Offs(pOrigin,82.82,-50.62,-0.00),v40,z0,tcp\WObj:=Plywood;
    MoveL Offs(pOrigin,82.57,-50.79,-0.00),v40,z0,tcp\WObj:=Plywood;
    MoveL Offs(pOrigin,81.97,-53.03,-0.00),v40,z0,tcp\WObj:=Plywood;
    MoveL Offs(pOrigin,82.36,-55.36,-0.00),v40,z0,tcp\WObj:=Plywood;
    MoveL Offs(pOrigin,87.42,-62.80,-0.00),v40,z0,tcp\WObj:=Plywood;
    MoveL Offs(pOrigin,89.65,-66.84,-0.00),v40,z0,tcp\WObj:=Plywood;
    MoveL Offs(pOrigin,91.43,-72.15,-0.00),v40,z0,tcp\WObj:=Plywood;
    MoveL Offs(pOrigin,91.96,-76.97,-0.00),v40,z0,tcp\WObj:=Plywood;
    MoveL Offs(pOrigin,91.00,-71.62,-0.00),v40,z0,tcp\WObj:=Plywood;
    MoveL Offs(pOrigin,89.02,-66.41,-0.00),v40,z0,tcp\WObj:=Plywood;
    MoveL Offs(pOrigin,81.86,-55.11,-0.00),v40,z0,tcp\WObj:=Plywood;
    MoveL Offs(pOrigin,81.76,-56.00,-0.00),v40,z0,tcp\WObj:=Plywood;
    MoveL Offs(pOrigin,82.68,-58.55,-0.00),v40,z0,tcp\WObj:=Plywood;
    MoveL Offs(pOrigin,85.83,-63.79,-0.00),v40,z0,tcp\WObj:=Plywood;
    MoveL Offs(pOrigin,83.10,-60.04,-0.00),v40,z0,tcp\WObj:=Plywood;
    MoveL Offs(pOrigin,81.54,-57.10,-0.00),v40,z0,tcp\WObj:=Plywood;
    MoveL Offs(pOrigin,79.74,-68.32,-0.00),v40,z0,tcp\WObj:=Plywood;
    MoveL Offs(pOrigin,74.00,-87.13,-0.00),v40,z0,tcp\WObj:=Plywood;
    MoveL Offs(pOrigin,72.62,-94.04,-0.00),v40,z0,tcp\WObj:=Plywood;
    MoveL Offs(pOrigin,72.72,-95.95,-0.00),v40,z0,tcp\WObj:=Plywood;
    MoveL Offs(pOrigin,73.36,-96.52,-0.00),v40,z0,tcp\WObj:=Plywood;
    MoveL Offs(pOrigin,87.49,-101.01,-0.00),v40,z0,tcp\WObj:=Plywood;
    MoveL Offs(pOrigin,100.99,-107.35,-0.00),v40,z0,tcp\WObj:=Plywood;
    MoveL Offs(pOrigin,107.57,-108.70,-0.00),v40,z0,tcp\WObj:=Plywood;
    MoveL Offs(pOrigin,107.68,-108.38,-0.00),v40,z0,tcp\WObj:=Plywood;
    MoveL Offs(pOrigin,105.56,-106.54,-0.00),v40,z0,tcp\WObj:=Plywood;
    MoveL Offs(pOrigin,97.80,-104.59,-0.00),v40,z0,tcp\WObj:=Plywood;
    MoveL Offs(pOrigin,88.88,-100.38,-0.00),v40,z0,tcp\WObj:=Plywood;
    MoveL Offs(pOrigin,80.02,-97.61,-0.00),v40,z0,tcp\WObj:=Plywood;
    MoveL Offs(pOrigin,88.13,-99.85,-0.00),v40,z0,tcp\WObj:=Plywood;
    MoveL Offs(pOrigin,98.54,-104.45,-0.00),v40,z0,tcp\WObj:=Plywood;
    MoveL Offs(pOrigin,101.62,-105.19,-0.00),v40,z0,tcp\WObj:=Plywood;
    MoveL Offs(pOrigin,104.95,-105.51,-0.00),v40,z0,tcp\WObj:=Plywood;
    MoveL Offs(pOrigin,98.22,-97.44,-0.00),v40,z0,tcp\WObj:=Plywood;
    MoveL Offs(pOrigin,98.44,-96.94,-0.00),v40,z0,tcp\WObj:=Plywood;
    MoveL Offs(pOrigin,103.54,-94.92,-0.00),v40,z0,tcp\WObj:=Plywood;
    MoveL Offs(pOrigin,97.27,-91.63,-0.00),v40,z0,tcp\WObj:=Plywood;
    MoveL Offs(pOrigin,96.91,-91.06,-0.00),v40,z0,tcp\WObj:=Plywood;
    MoveL Offs(pOrigin,103.22,-67.16,-0.00),v40,z0,tcp\WObj:=Plywood;
    MoveL Offs(pOrigin,105.24,-50.33,-0.00),v40,z0,tcp\WObj:=Plywood;
    MoveL Offs(pOrigin,104.07,-64.00,-0.00),v40,z0,tcp\WObj:=Plywood;
    MoveL Offs(pOrigin,107.15,-52.49,-0.00),v40,z0,tcp\WObj:=Plywood;
    MoveL Offs(pOrigin,108.32,-43.25,-0.00),v40,z0,tcp\WObj:=Plywood;
    MoveL Offs(pOrigin,108.43,-38.04,-0.00),v40,z0,tcp\WObj:=Plywood;
    MoveL Offs(pOrigin,108.00,-34.50,-0.00),v40,z0,tcp\WObj:=Plywood;
    MoveL Offs(pOrigin,107.89,-36.88,-0.00),v40,z0,tcp\WObj:=Plywood;
    MoveL Offs(pOrigin,106.94,-38.79,-0.00),v40,z0,tcp\WObj:=Plywood;
    MoveL Offs(pOrigin,103.75,-40.17,-0.00),v40,z0,tcp\WObj:=Plywood;
    MoveL Offs(pOrigin,97.38,-40.74,-0.00),v40,z0,tcp\WObj:=Plywood;
    MoveL Offs(pOrigin,95.18,-42.61,-0.00),v40,z0,tcp\WObj:=Plywood;
    MoveL Offs(pOrigin,94.82,-43.46,-0.00),v40,fine,tcp\WObj:=Plywood;
    MoveL Offs(pOrigin,94.82,-43.46,-6.00),v60,z5,tcp\WObj:=Plywood;
    MoveL Offs(pOrigin,94.86,-41.76,-6.00),vTravel,z5,tcp\WObj:=Plywood;
    MoveL Offs(pOrigin,94.86,-41.76,-0.00),v60,z0,tcp\WObj:=Plywood;
    MoveL Offs(pOrigin,96.31,-40.81,-0.00),v40,z0,tcp\WObj:=Plywood;
    MoveL Offs(pOrigin,97.91,-39.14,-0.00),v40,z0,tcp\WObj:=Plywood;
    MoveL Offs(pOrigin,96.63,-39.96,-0.00),v40,z0,tcp\WObj:=Plywood;
    MoveL Offs(pOrigin,94.86,-41.76,-0.00),v40,z0,tcp\WObj:=Plywood;
    MoveL Offs(pOrigin,94.72,-41.41,-0.00),v40,z0,tcp\WObj:=Plywood;
    MoveL Offs(pOrigin,95.96,-40.17,-0.00),v40,z0,tcp\WObj:=Plywood;
    MoveL Offs(pOrigin,94.29,-40.74,-0.00),v40,z0,tcp\WObj:=Plywood;
    MoveL Offs(pOrigin,94.22,-41.12,-0.00),v40,z0,tcp\WObj:=Plywood;
    MoveL Offs(pOrigin,94.72,-41.41,-0.00),v40,fine,tcp\WObj:=Plywood;
    MoveL Offs(pOrigin,94.72,-41.41,-6.00),v60,z5,tcp\WObj:=Plywood;
    MoveL Offs(pOrigin,98.26,-39.96,-6.00),vTravel,z5,tcp\WObj:=Plywood;
    MoveL Offs(pOrigin,98.26,-39.96,-0.00),v60,z0,tcp\WObj:=Plywood;
    MoveL Offs(pOrigin,102.90,-39.74,-0.00),v40,z0,tcp\WObj:=Plywood;
    MoveL Offs(pOrigin,106.09,-38.58,-0.00),v40,z0,tcp\WObj:=Plywood;
    MoveL Offs(pOrigin,107.15,-37.19,-0.00),v40,z0,tcp\WObj:=Plywood;
    MoveL Offs(pOrigin,107.43,-33.58,-0.00),v40,z0,tcp\WObj:=Plywood;
    MoveL Offs(pOrigin,102.79,-37.19,-0.00),v40,z0,tcp\WObj:=Plywood;
    MoveL Offs(pOrigin,102.94,-37.55,-0.00),v40,z0,tcp\WObj:=Plywood;
    MoveL Offs(pOrigin,102.47,-37.23,-0.00),v40,z0,tcp\WObj:=Plywood;
    MoveL Offs(pOrigin,100.03,-38.22,-0.00),v40,z0,tcp\WObj:=Plywood;
    MoveL Offs(pOrigin,98.26,-39.96,-0.00),v40,fine,tcp\WObj:=Plywood;
    MoveL Offs(pOrigin,98.26,-39.96,-6.00),v60,z5,tcp\WObj:=Plywood;
    MoveL Offs(pOrigin,109.06,-41.76,-6.00),vTravel,z5,tcp\WObj:=Plywood;
    MoveL Offs(pOrigin,109.06,-41.76,-0.00),v60,z0,tcp\WObj:=Plywood;
    MoveL Offs(pOrigin,108.64,-47.39,-0.00),v40,z0,tcp\WObj:=Plywood;
    MoveL Offs(pOrigin,107.68,-53.34,-0.00),v40,z0,tcp\WObj:=Plywood;
    MoveL Offs(pOrigin,97.59,-90.96,-0.00),v40,z0,tcp\WObj:=Plywood;
    MoveL Offs(pOrigin,105.98,-95.84,-0.00),v40,z0,tcp\WObj:=Plywood;
    MoveL Offs(pOrigin,110.97,-100.16,-0.00),v40,z0,tcp\WObj:=Plywood;
    MoveL Offs(pOrigin,112.89,-91.49,-0.00),v40,z0,tcp\WObj:=Plywood;
    MoveL Offs(pOrigin,114.48,-79.06,-0.00),v40,z0,tcp\WObj:=Plywood;
    MoveL Offs(pOrigin,115.65,-65.78,-0.00),v40,z0,tcp\WObj:=Plywood;
    MoveL Offs(pOrigin,115.76,-55.89,-0.00),v40,z0,tcp\WObj:=Plywood;
    MoveL Offs(pOrigin,115.22,-48.78,-0.00),v40,z0,tcp\WObj:=Plywood;
    MoveL Offs(pOrigin,113.95,-40.28,-0.00),v40,z0,tcp\WObj:=Plywood;
    MoveL Offs(pOrigin,111.93,-31.88,-0.00),v40,z0,tcp\WObj:=Plywood;
    MoveL Offs(pOrigin,110.44,-27.95,-0.00),v40,z0,tcp\WObj:=Plywood;
    MoveL Offs(pOrigin,108.89,-29.54,-0.00),v40,z0,tcp\WObj:=Plywood;
    MoveL Offs(pOrigin,109.06,-30.92,-0.00),v40,z0,tcp\WObj:=Plywood;
    MoveL Offs(pOrigin,108.53,-32.31,-0.00),v40,z0,tcp\WObj:=Plywood;
    MoveL Offs(pOrigin,108.96,-36.03,-0.00),v40,z0,tcp\WObj:=Plywood;
    MoveL Offs(pOrigin,109.06,-41.76,-0.00),v40,fine,tcp\WObj:=Plywood;
    MoveL Offs(pOrigin,109.06,-41.76,-6.00),v60,z5,tcp\WObj:=Plywood;
    MoveL Offs(pOrigin,115.26,-43.78,-6.00),vTravel,z5,tcp\WObj:=Plywood;
    MoveL Offs(pOrigin,115.26,-43.78,-0.00),v60,z0,tcp\WObj:=Plywood;
    MoveL Offs(pOrigin,118.34,-39.07,-0.00),v40,z0,tcp\WObj:=Plywood;
    MoveL Offs(pOrigin,116.15,-42.51,-0.00),v40,z0,tcp\WObj:=Plywood;
    MoveL Offs(pOrigin,115.33,-44.63,-0.00),v40,z0,tcp\WObj:=Plywood;
    MoveL Offs(pOrigin,116.39,-55.04,-0.00),v40,z0,tcp\WObj:=Plywood;
    MoveL Offs(pOrigin,116.39,-63.54,-0.00),v40,z0,tcp\WObj:=Plywood;
    MoveL Offs(pOrigin,114.38,-85.89,-0.00),v40,z0,tcp\WObj:=Plywood;
    MoveL Offs(pOrigin,119.37,-74.35,-0.00),v40,z0,tcp\WObj:=Plywood;
    MoveL Offs(pOrigin,114.16,-87.77,-0.00),v40,z0,tcp\WObj:=Plywood;
    MoveL Offs(pOrigin,114.84,-91.91,-0.00),v40,z0,tcp\WObj:=Plywood;
    MoveL Offs(pOrigin,119.16,-87.45,-0.00),v40,z0,tcp\WObj:=Plywood;
    MoveL Offs(pOrigin,121.95,-85.40,-0.00),v40,z0,tcp\WObj:=Plywood;
    MoveL Offs(pOrigin,117.78,-88.94,-0.00),v40,z0,tcp\WObj:=Plywood;
    MoveL Offs(pOrigin,114.84,-92.23,-0.00),v40,z0,tcp\WObj:=Plywood;
    MoveL Offs(pOrigin,115.12,-95.21,-0.00),v40,z0,tcp\WObj:=Plywood;
    MoveL Offs(pOrigin,115.97,-96.20,-0.00),v40,z0,tcp\WObj:=Plywood;
  ENDPROC

  PROC DrawPart8()
    MoveL Offs(pOrigin,117.35,-95.74,-0.00),v40,z0,tcp\WObj:=Plywood;
    MoveL Offs(pOrigin,118.80,-93.90,-0.00),v40,z0,tcp\WObj:=Plywood;
    MoveL Offs(pOrigin,117.78,-95.53,-0.00),v40,z0,tcp\WObj:=Plywood;
    MoveL Offs(pOrigin,116.71,-96.52,-0.00),v40,z0,tcp\WObj:=Plywood;
    MoveL Offs(pOrigin,115.54,-96.52,-0.00),v40,z0,tcp\WObj:=Plywood;
    MoveL Offs(pOrigin,114.66,-95.42,-0.00),v40,z0,tcp\WObj:=Plywood;
    MoveL Offs(pOrigin,114.16,-90.32,-0.00),v40,z0,tcp\WObj:=Plywood;
    MoveL Offs(pOrigin,113.77,-89.47,-0.00),v40,z0,tcp\WObj:=Plywood;
    MoveL Offs(pOrigin,111.08,-102.86,-0.00),v40,z0,tcp\WObj:=Plywood;
    MoveL Offs(pOrigin,110.55,-107.07,-0.00),v40,z0,tcp\WObj:=Plywood;
    MoveL Offs(pOrigin,112.57,-105.09,-0.00),v40,z0,tcp\WObj:=Plywood;
    MoveL Offs(pOrigin,115.40,-100.20,-0.00),v40,z0,tcp\WObj:=Plywood;
    MoveL Offs(pOrigin,119.30,-94.68,-0.00),v40,z0,tcp\WObj:=Plywood;
    MoveL Offs(pOrigin,120.79,-91.91,-0.00),v40,z0,tcp\WObj:=Plywood;
    MoveL Offs(pOrigin,122.66,-87.13,-0.00),v40,z0,tcp\WObj:=Plywood;
    MoveL Offs(pOrigin,126.13,-84.26,-0.00),v40,z0,tcp\WObj:=Plywood;
    MoveL Offs(pOrigin,123.58,-80.76,-0.00),v40,z0,tcp\WObj:=Plywood;
    MoveL Offs(pOrigin,122.56,-76.29,-0.00),v40,z0,tcp\WObj:=Plywood;
    MoveL Offs(pOrigin,121.39,-47.82,-0.00),v40,z0,tcp\WObj:=Plywood;
    MoveL Offs(pOrigin,119.05,-22.74,-0.00),v40,z0,tcp\WObj:=Plywood;
    MoveL Offs(pOrigin,113.84,-23.10,-0.00),v40,z0,tcp\WObj:=Plywood;
    MoveL Offs(pOrigin,111.08,-27.31,-0.00),v40,z0,tcp\WObj:=Plywood;
    MoveL Offs(pOrigin,113.53,-35.17,-0.00),v40,z0,tcp\WObj:=Plywood;
    MoveL Offs(pOrigin,117.49,-29.61,-0.00),v40,z0,tcp\WObj:=Plywood;
    MoveL Offs(pOrigin,113.70,-35.28,-0.00),v40,z0,tcp\WObj:=Plywood;
    MoveL Offs(pOrigin,113.74,-35.99,-0.00),v40,z0,tcp\WObj:=Plywood;
    MoveL Offs(pOrigin,116.39,-34.89,-0.00),v40,z0,tcp\WObj:=Plywood;
    MoveL Offs(pOrigin,118.13,-33.62,-0.00),v40,z0,tcp\WObj:=Plywood;
    MoveL Offs(pOrigin,116.50,-35.00,-0.00),v40,z0,tcp\WObj:=Plywood;
    MoveL Offs(pOrigin,113.77,-36.34,-0.00),v40,z0,tcp\WObj:=Plywood;
    MoveL Offs(pOrigin,115.26,-43.78,-0.00),v40,fine,tcp\WObj:=Plywood;
    MoveL Offs(pOrigin,115.26,-43.78,-6.00),v60,z5,tcp\WObj:=Plywood;
    MoveL Offs(pOrigin,121.07,-40.06,-6.00),vTravel,z5,tcp\WObj:=Plywood;
    MoveL Offs(pOrigin,121.07,-40.06,-0.00),v60,z0,tcp\WObj:=Plywood;
    MoveL Offs(pOrigin,121.81,-50.90,-0.00),v40,z0,tcp\WObj:=Plywood;
    MoveL Offs(pOrigin,122.56,-73.32,-0.00),v40,z0,tcp\WObj:=Plywood;
    MoveL Offs(pOrigin,123.41,-79.27,-0.00),v40,z0,tcp\WObj:=Plywood;
    MoveL Offs(pOrigin,125.00,-82.24,-0.00),v40,z0,tcp\WObj:=Plywood;
    MoveL Offs(pOrigin,129.92,-87.24,-0.00),v40,z0,tcp\WObj:=Plywood;
    MoveL Offs(pOrigin,130.81,-90.21,-0.00),v40,z0,tcp\WObj:=Plywood;
    MoveL Offs(pOrigin,137.25,-99.78,-0.00),v40,z0,tcp\WObj:=Plywood;
    MoveL Offs(pOrigin,140.65,-105.62,-0.00),v40,z0,tcp\WObj:=Plywood;
    MoveL Offs(pOrigin,144.12,-113.52,-0.00),v40,z0,tcp\WObj:=Plywood;
    MoveL Offs(pOrigin,144.34,-109.55,-0.00),v40,z0,tcp\WObj:=Plywood;
    MoveL Offs(pOrigin,143.81,-105.51,-0.00),v40,z0,tcp\WObj:=Plywood;
    MoveL Offs(pOrigin,140.26,-90.85,-0.00),v40,z0,tcp\WObj:=Plywood;
    MoveL Offs(pOrigin,139.77,-91.49,-0.00),v40,z0,tcp\WObj:=Plywood;
    MoveL Offs(pOrigin,138.74,-95.74,-0.00),v40,z0,tcp\WObj:=Plywood;
    MoveL Offs(pOrigin,138.18,-96.59,-0.00),v40,z0,tcp\WObj:=Plywood;
    MoveL Offs(pOrigin,137.22,-97.01,-0.00),v40,z0,tcp\WObj:=Plywood;
    MoveL Offs(pOrigin,136.05,-96.38,-0.00),v40,z0,tcp\WObj:=Plywood;
    MoveL Offs(pOrigin,133.43,-91.91,-0.00),v40,z0,tcp\WObj:=Plywood;
    MoveL Offs(pOrigin,135.94,-95.74,-0.00),v40,z0,tcp\WObj:=Plywood;
    MoveL Offs(pOrigin,136.79,-96.52,-0.00),v40,z0,tcp\WObj:=Plywood;
    MoveL Offs(pOrigin,137.54,-96.45,-0.00),v40,z0,tcp\WObj:=Plywood;
    MoveL Offs(pOrigin,138.32,-95.42,-0.00),v40,z0,tcp\WObj:=Plywood;
    MoveL Offs(pOrigin,138.67,-93.40,-0.00),v40,z0,tcp\WObj:=Plywood;
    MoveL Offs(pOrigin,134.10,-90.53,-0.00),v40,z0,tcp\WObj:=Plywood;
    MoveL Offs(pOrigin,138.71,-93.15,-0.00),v40,z0,tcp\WObj:=Plywood;
    MoveL Offs(pOrigin,139.91,-89.47,-0.00),v40,z0,tcp\WObj:=Plywood;
    MoveL Offs(pOrigin,138.07,-80.76,-0.00),v40,z0,tcp\WObj:=Plywood;
    MoveL Offs(pOrigin,134.35,-71.19,-0.00),v40,z0,tcp\WObj:=Plywood;
    MoveL Offs(pOrigin,137.54,-78.45,-0.00),v40,z0,tcp\WObj:=Plywood;
    MoveL Offs(pOrigin,135.94,-67.16,-0.00),v40,z0,tcp\WObj:=Plywood;
    MoveL Offs(pOrigin,135.31,-60.14,-0.00),v40,z0,tcp\WObj:=Plywood;
    MoveL Offs(pOrigin,135.31,-50.79,-0.00),v40,z0,tcp\WObj:=Plywood;
    MoveL Offs(pOrigin,136.05,-43.14,-0.00),v40,z0,tcp\WObj:=Plywood;
    MoveL Offs(pOrigin,134.14,-40.06,-0.00),v40,z0,tcp\WObj:=Plywood;
    MoveL Offs(pOrigin,130.49,-35.88,-0.00),v40,z0,tcp\WObj:=Plywood;
    MoveL Offs(pOrigin,133.93,-39.42,-0.00),v40,z0,tcp\WObj:=Plywood;
    MoveL Offs(pOrigin,136.05,-42.44,-0.00),v40,z0,tcp\WObj:=Plywood;
    MoveL Offs(pOrigin,137.32,-35.49,-0.00),v40,z0,tcp\WObj:=Plywood;
    MoveL Offs(pOrigin,129.57,-31.67,-0.00),v40,z0,tcp\WObj:=Plywood;
    MoveL Offs(pOrigin,124.26,-26.67,-0.00),v40,z0,tcp\WObj:=Plywood;
    MoveL Offs(pOrigin,121.18,-22.74,-0.00),v40,z0,tcp\WObj:=Plywood;
    MoveL Offs(pOrigin,119.79,-22.64,-0.00),v40,z0,tcp\WObj:=Plywood;
    MoveL Offs(pOrigin,119.47,-22.96,-0.00),v40,z0,tcp\WObj:=Plywood;
    MoveL Offs(pOrigin,121.07,-40.06,-0.00),v40,fine,tcp\WObj:=Plywood;
    MoveL Offs(pOrigin,121.07,-40.06,-6.00),v60,z5,tcp\WObj:=Plywood;
    MoveL Offs(pOrigin,122.95,-37.41,-6.00),vTravel,z5,tcp\WObj:=Plywood;
    MoveL Offs(pOrigin,122.95,-37.41,-0.00),v60,z0,tcp\WObj:=Plywood;
    MoveL Offs(pOrigin,122.77,-36.34,-0.00),v40,z0,tcp\WObj:=Plywood;
    MoveL Offs(pOrigin,123.30,-35.49,-0.00),v40,z0,tcp\WObj:=Plywood;
    MoveL Offs(pOrigin,124.36,-35.17,-0.00),v40,z0,tcp\WObj:=Plywood;
    MoveL Offs(pOrigin,125.39,-35.71,-0.00),v40,z0,tcp\WObj:=Plywood;
    MoveL Offs(pOrigin,125.74,-36.98,-0.00),v40,z0,tcp\WObj:=Plywood;
    MoveL Offs(pOrigin,125.00,-37.97,-0.00),v40,z0,tcp\WObj:=Plywood;
    MoveL Offs(pOrigin,123.94,-38.15,-0.00),v40,z0,tcp\WObj:=Plywood;
    MoveL Offs(pOrigin,122.95,-37.41,-0.00),v40,z0,tcp\WObj:=Plywood;
    MoveL Offs(pOrigin,123.19,-37.51,-0.00),v40,z0,tcp\WObj:=Plywood;
    MoveL Offs(pOrigin,124.04,-38.04,-0.00),v40,z0,tcp\WObj:=Plywood;
    MoveL Offs(pOrigin,124.89,-37.87,-0.00),v40,z0,tcp\WObj:=Plywood;
    MoveL Offs(pOrigin,125.53,-37.09,-0.00),v40,z0,tcp\WObj:=Plywood;
    MoveL Offs(pOrigin,125.46,-36.13,-0.00),v40,z0,tcp\WObj:=Plywood;
    MoveL Offs(pOrigin,124.47,-35.39,-0.00),v40,z0,tcp\WObj:=Plywood;
    MoveL Offs(pOrigin,123.30,-35.74,-0.00),v40,z0,tcp\WObj:=Plywood;
    MoveL Offs(pOrigin,122.88,-36.56,-0.00),v40,z0,tcp\WObj:=Plywood;
    MoveL Offs(pOrigin,123.19,-37.51,-0.00),v40,fine,tcp\WObj:=Plywood;
    MoveL Offs(pOrigin,123.19,-37.51,-6.00),v60,z5,tcp\WObj:=Plywood;
    MoveL Offs(pOrigin,127.48,-45.45,-6.00),vTravel,z5,tcp\WObj:=Plywood;
    MoveL Offs(pOrigin,127.48,-45.45,-0.00),v60,z0,tcp\WObj:=Plywood;
    MoveL Offs(pOrigin,130.77,-51.22,-0.00),v40,z0,tcp\WObj:=Plywood;
    MoveL Offs(pOrigin,134.35,-59.97,-0.00),v40,z0,tcp\WObj:=Plywood;
    MoveL Offs(pOrigin,131.09,-52.39,-0.00),v40,z0,tcp\WObj:=Plywood;
    MoveL Offs(pOrigin,127.48,-45.45,-0.00),v40,fine,tcp\WObj:=Plywood;
    MoveL Offs(pOrigin,127.48,-45.45,-6.00),v60,z5,tcp\WObj:=Plywood;
    MoveL Offs(pOrigin,133.85,-42.12,-6.00),vTravel,z5,tcp\WObj:=Plywood;
    MoveL Offs(pOrigin,133.85,-42.12,-0.00),v60,z0,tcp\WObj:=Plywood;
    MoveL Offs(pOrigin,131.76,-39.39,-0.00),v40,z0,tcp\WObj:=Plywood;
    MoveL Offs(pOrigin,133.85,-42.12,-0.00),v40,fine,tcp\WObj:=Plywood;
    MoveL Offs(pOrigin,133.85,-42.12,-6.00),v60,z5,tcp\WObj:=Plywood;
    MoveL Offs(pOrigin,137.01,-41.02,-6.00),vTravel,z5,tcp\WObj:=Plywood;
    MoveL Offs(pOrigin,137.01,-41.02,-0.00),v60,z0,tcp\WObj:=Plywood;
    MoveL Offs(pOrigin,136.05,-49.94,-0.00),v40,z0,tcp\WObj:=Plywood;
    MoveL Offs(pOrigin,135.94,-59.51,-0.00),v40,z0,tcp\WObj:=Plywood;
    MoveL Offs(pOrigin,137.22,-72.04,-0.00),v40,z0,tcp\WObj:=Plywood;
    MoveL Offs(pOrigin,139.34,-84.16,-0.00),v40,z0,tcp\WObj:=Plywood;
    MoveL Offs(pOrigin,143.27,-100.73,-0.00),v40,z0,tcp\WObj:=Plywood;
    MoveL Offs(pOrigin,143.81,-101.76,-0.00),v40,z0,tcp\WObj:=Plywood;
    MoveL Offs(pOrigin,150.39,-96.66,-0.00),v40,z0,tcp\WObj:=Plywood;
  ENDPROC

  PROC DrawPart9()
    MoveL Offs(pOrigin,158.36,-93.68,-0.00),v40,z0,tcp\WObj:=Plywood;
    MoveL Offs(pOrigin,158.57,-93.19,-0.00),v40,z0,tcp\WObj:=Plywood;
    MoveL Offs(pOrigin,145.82,-53.03,-0.00),v40,z0,tcp\WObj:=Plywood;
    MoveL Offs(pOrigin,143.49,-43.14,-0.00),v40,z0,tcp\WObj:=Plywood;
    MoveL Offs(pOrigin,142.50,-36.77,-0.00),v40,z0,tcp\WObj:=Plywood;
    MoveL Offs(pOrigin,140.62,-36.66,-0.00),v40,z0,tcp\WObj:=Plywood;
    MoveL Offs(pOrigin,138.18,-35.71,-0.00),v40,z0,tcp\WObj:=Plywood;
    MoveL Offs(pOrigin,137.86,-36.03,-0.00),v40,z0,tcp\WObj:=Plywood;
    MoveL Offs(pOrigin,137.01,-41.02,-0.00),v40,fine,tcp\WObj:=Plywood;
    MoveL Offs(pOrigin,137.01,-41.02,-6.00),v60,z5,tcp\WObj:=Plywood;
    MoveL Offs(pOrigin,141.04,-36.13,-6.00),vTravel,z5,tcp\WObj:=Plywood;
    MoveL Offs(pOrigin,141.04,-36.13,-0.00),v60,z0,tcp\WObj:=Plywood;
    MoveL Offs(pOrigin,142.64,-35.95,-0.00),v40,z0,tcp\WObj:=Plywood;
    MoveL Offs(pOrigin,145.72,-34.29,-0.00),v40,z0,tcp\WObj:=Plywood;
    MoveL Offs(pOrigin,150.82,-32.62,-0.00),v40,z0,tcp\WObj:=Plywood;
    MoveL Offs(pOrigin,152.62,-32.31,-0.00),v40,z0,tcp\WObj:=Plywood;
    MoveL Offs(pOrigin,156.45,-32.62,-0.00),v40,z0,tcp\WObj:=Plywood;
    MoveL Offs(pOrigin,157.30,-32.34,-0.00),v40,z0,tcp\WObj:=Plywood;
    MoveL Offs(pOrigin,160.31,-29.33,-0.00),v40,z0,tcp\WObj:=Plywood;
    MoveL Offs(pOrigin,161.23,-27.31,-0.00),v40,z0,tcp\WObj:=Plywood;
    MoveL Offs(pOrigin,161.76,-24.55,-0.00),v40,z0,tcp\WObj:=Plywood;
    MoveL Offs(pOrigin,161.55,-20.94,-0.00),v40,z0,tcp\WObj:=Plywood;
    MoveL Offs(pOrigin,160.49,-18.92,-0.00),v40,z0,tcp\WObj:=Plywood;
    MoveL Offs(pOrigin,156.13,-16.65,-0.00),v40,z0,tcp\WObj:=Plywood;
    MoveL Offs(pOrigin,151.77,-15.41,-0.00),v40,z0,tcp\WObj:=Plywood;
    MoveL Offs(pOrigin,147.63,-15.62,-0.00),v40,z0,tcp\WObj:=Plywood;
    MoveL Offs(pOrigin,148.91,-16.83,-0.00),v40,z0,tcp\WObj:=Plywood;
    MoveL Offs(pOrigin,146.57,-15.77,-0.00),v40,z0,tcp\WObj:=Plywood;
    MoveL Offs(pOrigin,142.11,-14.56,-0.00),v40,z0,tcp\WObj:=Plywood;
    MoveL Offs(pOrigin,139.45,-14.56,-0.00),v40,z0,tcp\WObj:=Plywood;
    MoveL Offs(pOrigin,138.07,-15.31,-0.00),v40,z0,tcp\WObj:=Plywood;
    MoveL Offs(pOrigin,137.22,-17.01,-0.00),v40,z0,tcp\WObj:=Plywood;
    MoveL Offs(pOrigin,137.43,-17.57,-0.00),v40,z0,tcp\WObj:=Plywood;
    MoveL Offs(pOrigin,147.10,-21.29,-0.00),v40,z0,tcp\WObj:=Plywood;
    MoveL Offs(pOrigin,147.28,-21.75,-0.00),v40,z0,tcp\WObj:=Plywood;
    MoveL Offs(pOrigin,145.86,-21.47,-0.00),v40,z0,tcp\WObj:=Plywood;
    MoveL Offs(pOrigin,145.82,-22.96,-0.00),v40,z0,tcp\WObj:=Plywood;
    MoveL Offs(pOrigin,144.76,-25.61,-0.00),v40,z0,tcp\WObj:=Plywood;
    MoveL Offs(pOrigin,143.17,-25.97,-0.00),v40,z0,tcp\WObj:=Plywood;
    MoveL Offs(pOrigin,144.37,-26.75,-0.00),v40,z0,tcp\WObj:=Plywood;
    MoveL Offs(pOrigin,144.02,-26.99,-0.00),v40,z0,tcp\WObj:=Plywood;
    MoveL Offs(pOrigin,138.07,-24.80,-0.00),v40,z0,tcp\WObj:=Plywood;
    MoveL Offs(pOrigin,129.25,-20.44,-0.00),v40,z0,tcp\WObj:=Plywood;
    MoveL Offs(pOrigin,126.17,-18.35,-0.00),v40,z0,tcp\WObj:=Plywood;
    MoveL Offs(pOrigin,125.00,-17.96,-0.00),v40,z0,tcp\WObj:=Plywood;
    MoveL Offs(pOrigin,123.72,-18.03,-0.00),v40,z0,tcp\WObj:=Plywood;
    MoveL Offs(pOrigin,123.09,-18.39,-0.00),v40,z0,tcp\WObj:=Plywood;
    MoveL Offs(pOrigin,122.63,-19.66,-0.00),v40,z0,tcp\WObj:=Plywood;
    MoveL Offs(pOrigin,123.62,-21.36,-0.00),v40,z0,tcp\WObj:=Plywood;
    MoveL Offs(pOrigin,131.27,-27.14,-0.00),v40,z0,tcp\WObj:=Plywood;
    MoveL Offs(pOrigin,134.35,-28.84,-0.00),v40,z0,tcp\WObj:=Plywood;
    MoveL Offs(pOrigin,139.02,-30.57,-0.00),v40,z0,tcp\WObj:=Plywood;
    MoveL Offs(pOrigin,140.73,-31.60,-0.00),v40,z0,tcp\WObj:=Plywood;
    MoveL Offs(pOrigin,141.11,-32.24,-0.00),v40,z0,tcp\WObj:=Plywood;
    MoveL Offs(pOrigin,139.24,-31.10,-0.00),v40,z0,tcp\WObj:=Plywood;
    MoveL Offs(pOrigin,137.22,-30.50,-0.00),v40,z0,tcp\WObj:=Plywood;
    MoveL Offs(pOrigin,135.45,-33.69,-0.00),v40,z0,tcp\WObj:=Plywood;
    MoveL Offs(pOrigin,141.04,-36.13,-0.00),v40,fine,tcp\WObj:=Plywood;
    MoveL Offs(pOrigin,141.04,-36.13,-6.00),v60,z5,tcp\WObj:=Plywood;
    MoveL Offs(pOrigin,143.17,-36.56,-6.00),vTravel,z5,tcp\WObj:=Plywood;
    MoveL Offs(pOrigin,143.17,-36.56,-0.00),v60,z0,tcp\WObj:=Plywood;
    MoveL Offs(pOrigin,144.12,-42.93,-0.00),v40,z0,tcp\WObj:=Plywood;
    MoveL Offs(pOrigin,146.14,-51.15,-0.00),v40,z0,tcp\WObj:=Plywood;
    MoveL Offs(pOrigin,145.93,-42.40,-0.00),v40,z0,tcp\WObj:=Plywood;
    MoveL Offs(pOrigin,146.36,-38.79,-0.00),v40,z0,tcp\WObj:=Plywood;
    MoveL Offs(pOrigin,147.21,-35.35,-0.00),v40,z0,tcp\WObj:=Plywood;
    MoveL Offs(pOrigin,146.14,-42.93,-0.00),v40,z0,tcp\WObj:=Plywood;
    MoveL Offs(pOrigin,146.36,-51.54,-0.00),v40,z0,tcp\WObj:=Plywood;
    MoveL Offs(pOrigin,147.06,-54.83,-0.00),v40,z0,tcp\WObj:=Plywood;
    MoveL Offs(pOrigin,147.31,-55.11,-0.00),v40,z0,tcp\WObj:=Plywood;
    MoveL Offs(pOrigin,151.14,-55.79,-0.00),v40,z0,tcp\WObj:=Plywood;
    MoveL Offs(pOrigin,163.36,-58.87,-0.00),v40,z0,tcp\WObj:=Plywood;
    MoveL Offs(pOrigin,172.49,-61.70,-0.00),v40,z0,tcp\WObj:=Plywood;
    MoveL Offs(pOrigin,172.81,-62.48,-0.00),v40,z0,tcp\WObj:=Plywood;
    MoveL Offs(pOrigin,172.60,-67.47,-0.00),v40,z0,tcp\WObj:=Plywood;
    MoveL Offs(pOrigin,172.07,-67.58,-0.00),v40,z0,tcp\WObj:=Plywood;
    MoveL Offs(pOrigin,167.04,-66.20,-0.00),v40,z0,tcp\WObj:=Plywood;
    MoveL Offs(pOrigin,173.70,-71.44,-0.00),v40,z0,tcp\WObj:=Plywood;
    MoveL Offs(pOrigin,169.84,-68.96,-0.00),v40,z0,tcp\WObj:=Plywood;
    MoveL Offs(pOrigin,166.33,-65.92,-0.00),v40,z0,tcp\WObj:=Plywood;
    MoveL Offs(pOrigin,149.15,-61.21,-0.00),v40,z0,tcp\WObj:=Plywood;
    MoveL Offs(pOrigin,159.32,-93.51,-0.00),v40,z0,tcp\WObj:=Plywood;
    MoveL Offs(pOrigin,159.00,-94.07,-0.00),v40,z0,tcp\WObj:=Plywood;
    MoveL Offs(pOrigin,151.81,-96.69,-0.00),v40,z0,tcp\WObj:=Plywood;
    MoveL Offs(pOrigin,157.80,-99.78,-0.00),v40,z0,tcp\WObj:=Plywood;
    MoveL Offs(pOrigin,157.62,-100.41,-0.00),v40,z0,tcp\WObj:=Plywood;
    MoveL Offs(pOrigin,154.54,-104.56,-0.00),v40,z0,tcp\WObj:=Plywood;
    MoveL Offs(pOrigin,158.89,-103.71,-0.00),v40,z0,tcp\WObj:=Plywood;
    MoveL Offs(pOrigin,167.11,-101.05,-0.00),v40,z0,tcp\WObj:=Plywood;
    MoveL Offs(pOrigin,159.11,-104.03,-0.00),v40,z0,tcp\WObj:=Plywood;
    MoveL Offs(pOrigin,154.01,-105.12,-0.00),v40,z0,tcp\WObj:=Plywood;
    MoveL Offs(pOrigin,151.46,-108.17,-0.00),v40,z0,tcp\WObj:=Plywood;
    MoveL Offs(pOrigin,151.67,-108.38,-0.00),v40,z0,tcp\WObj:=Plywood;
    MoveL Offs(pOrigin,158.04,-106.50,-0.00),v40,z0,tcp\WObj:=Plywood;
    MoveL Offs(pOrigin,168.46,-102.18,-0.00),v40,z0,tcp\WObj:=Plywood;
    MoveL Offs(pOrigin,183.65,-97.86,-0.00),v40,z0,tcp\WObj:=Plywood;
    MoveL Offs(pOrigin,185.00,-97.12,-0.00),v40,z0,tcp\WObj:=Plywood;
    MoveL Offs(pOrigin,183.08,-93.82,-0.00),v40,z0,tcp\WObj:=Plywood;
    MoveL Offs(pOrigin,180.14,-84.58,-0.00),v40,z0,tcp\WObj:=Plywood;
    MoveL Offs(pOrigin,176.96,-71.94,-0.00),v40,z0,tcp\WObj:=Plywood;
    MoveL Offs(pOrigin,174.51,-59.83,-0.00),v40,z0,tcp\WObj:=Plywood;
    MoveL Offs(pOrigin,173.24,-55.36,-0.00),v40,z0,tcp\WObj:=Plywood;
    MoveL Offs(pOrigin,170.94,-48.99,-0.00),v40,z0,tcp\WObj:=Plywood;
    MoveL Offs(pOrigin,167.61,-41.23,-0.00),v40,z0,tcp\WObj:=Plywood;
    MoveL Offs(pOrigin,169.77,-45.48,-0.00),v40,z0,tcp\WObj:=Plywood;
    MoveL Offs(pOrigin,173.56,-54.76,-0.00),v40,z0,tcp\WObj:=Plywood;
    MoveL Offs(pOrigin,172.28,-48.99,-0.00),v40,z0,tcp\WObj:=Plywood;
    MoveL Offs(pOrigin,168.81,-40.28,-0.00),v40,z0,tcp\WObj:=Plywood;
    MoveL Offs(pOrigin,168.35,-39.96,-0.00),v40,z0,tcp\WObj:=Plywood;
    MoveL Offs(pOrigin,159.32,-38.26,-0.00),v40,z0,tcp\WObj:=Plywood;
    MoveL Offs(pOrigin,157.09,-37.44,-0.00),v40,z0,tcp\WObj:=Plywood;
    MoveL Offs(pOrigin,155.07,-36.17,-0.00),v40,z0,tcp\WObj:=Plywood;
    MoveL Offs(pOrigin,150.61,-34.89,-0.00),v40,z0,tcp\WObj:=Plywood;
    MoveL Offs(pOrigin,149.01,-33.79,-0.00),v40,z0,tcp\WObj:=Plywood;
    MoveL Offs(pOrigin,145.82,-34.93,-0.00),v40,z0,tcp\WObj:=Plywood;
    MoveL Offs(pOrigin,143.17,-36.56,-0.00),v40,fine,tcp\WObj:=Plywood;
    MoveL Offs(pOrigin,143.17,-36.56,-6.00),v60,z5,tcp\WObj:=Plywood;
    MoveL Offs(pOrigin,150.00,-33.69,-6.00),vTravel,z5,tcp\WObj:=Plywood;
    MoveL Offs(pOrigin,150.00,-33.69,-0.00),v60,z0,tcp\WObj:=Plywood;
    MoveL Offs(pOrigin,151.24,-34.47,-0.00),v40,z0,tcp\WObj:=Plywood;
  ENDPROC

  PROC DrawPart10()
    MoveL Offs(pOrigin,153.48,-35.17,-0.00),v40,z0,tcp\WObj:=Plywood;
    MoveL Offs(pOrigin,159.74,-36.24,-0.00),v40,z0,tcp\WObj:=Plywood;
    MoveL Offs(pOrigin,162.29,-35.74,-0.00),v40,z0,tcp\WObj:=Plywood;
    MoveL Offs(pOrigin,165.27,-34.36,-0.00),v40,z0,tcp\WObj:=Plywood;
    MoveL Offs(pOrigin,168.03,-32.31,-0.00),v40,z0,tcp\WObj:=Plywood;
    MoveL Offs(pOrigin,169.84,-30.50,-0.00),v40,z0,tcp\WObj:=Plywood;
    MoveL Offs(pOrigin,173.27,-25.51,-0.00),v40,z0,tcp\WObj:=Plywood;
    MoveL Offs(pOrigin,173.98,-23.06,-0.00),v40,z0,tcp\WObj:=Plywood;
    MoveL Offs(pOrigin,173.06,-19.77,-0.00),v40,z0,tcp\WObj:=Plywood;
    MoveL Offs(pOrigin,171.54,-18.14,-0.00),v40,z0,tcp\WObj:=Plywood;
    MoveL Offs(pOrigin,169.20,-17.22,-0.00),v40,z0,tcp\WObj:=Plywood;
    MoveL Offs(pOrigin,160.70,-15.62,-0.00),v40,z0,tcp\WObj:=Plywood;
    MoveL Offs(pOrigin,159.00,-15.66,-0.00),v40,z0,tcp\WObj:=Plywood;
    MoveL Offs(pOrigin,158.89,-15.91,-0.00),v40,z0,tcp\WObj:=Plywood;
    MoveL Offs(pOrigin,160.06,-16.23,-0.00),v40,z0,tcp\WObj:=Plywood;
    MoveL Offs(pOrigin,161.05,-17.33,-0.00),v40,z0,tcp\WObj:=Plywood;
    MoveL Offs(pOrigin,162.29,-21.47,-0.00),v40,z0,tcp\WObj:=Plywood;
    MoveL Offs(pOrigin,162.19,-25.72,-0.00),v40,z0,tcp\WObj:=Plywood;
    MoveL Offs(pOrigin,160.95,-29.97,-0.00),v40,z0,tcp\WObj:=Plywood;
    MoveL Offs(pOrigin,159.53,-32.20,-0.00),v40,z0,tcp\WObj:=Plywood;
    MoveL Offs(pOrigin,157.09,-33.94,-0.00),v40,z0,tcp\WObj:=Plywood;
    MoveL Offs(pOrigin,154.01,-34.54,-0.00),v40,z0,tcp\WObj:=Plywood;
    MoveL Offs(pOrigin,152.52,-34.33,-0.00),v40,z0,tcp\WObj:=Plywood;
    MoveL Offs(pOrigin,150.39,-33.44,-0.00),v40,z0,tcp\WObj:=Plywood;
    MoveL Offs(pOrigin,150.00,-33.69,-0.00),v40,fine,tcp\WObj:=Plywood;
    MoveL Offs(pOrigin,150.00,-33.69,-6.00),v60,z5,tcp\WObj:=Plywood;
    MoveL Offs(pOrigin,151.31,-33.26,-6.00),vTravel,z5,tcp\WObj:=Plywood;
    MoveL Offs(pOrigin,151.31,-33.26,-0.00),v60,z0,tcp\WObj:=Plywood;
    MoveL Offs(pOrigin,153.26,-33.90,-0.00),v40,z0,tcp\WObj:=Plywood;
    MoveL Offs(pOrigin,155.10,-33.69,-0.00),v40,z0,tcp\WObj:=Plywood;
    MoveL Offs(pOrigin,153.05,-32.94,-0.00),v40,z0,tcp\WObj:=Plywood;
    MoveL Offs(pOrigin,151.31,-33.26,-0.00),v40,fine,tcp\WObj:=Plywood;
    MoveL Offs(pOrigin,151.31,-33.26,-6.00),v60,z5,tcp\WObj:=Plywood;
    MoveL Offs(pOrigin,155.67,-33.26,-6.00),vTravel,z5,tcp\WObj:=Plywood;
    MoveL Offs(pOrigin,155.67,-33.26,-0.00),v60,z0,tcp\WObj:=Plywood;
    MoveL Offs(pOrigin,156.84,-33.37,-0.00),v40,z0,tcp\WObj:=Plywood;
    MoveL Offs(pOrigin,155.67,-33.26,-0.00),v40,fine,tcp\WObj:=Plywood;
    MoveL Offs(pOrigin,155.67,-33.26,-6.00),v60,z5,tcp\WObj:=Plywood;
    MoveL Offs(pOrigin,157.09,-32.70,-6.00),vTravel,z5,tcp\WObj:=Plywood;
    MoveL Offs(pOrigin,157.09,-32.70,-0.00),v60,z0,tcp\WObj:=Plywood;
    MoveL Offs(pOrigin,158.26,-32.52,-0.00),v40,z0,tcp\WObj:=Plywood;
    MoveL Offs(pOrigin,159.21,-31.56,-0.00),v40,z0,tcp\WObj:=Plywood;
    MoveL Offs(pOrigin,160.24,-29.76,-0.00),v40,z0,tcp\WObj:=Plywood;
    MoveL Offs(pOrigin,157.09,-32.70,-0.00),v40,fine,tcp\WObj:=Plywood;
    MoveL Offs(pOrigin,157.09,-32.70,-6.00),v60,z5,tcp\WObj:=Plywood;
    MoveL Offs(pOrigin,158.75,-30.64,-6.00),vTravel,z5,tcp\WObj:=Plywood;
    MoveL Offs(pOrigin,158.75,-30.64,-0.00),v60,z0,tcp\WObj:=Plywood;
    MoveL Offs(pOrigin,160.81,-26.67,-0.00),v40,z0,tcp\WObj:=Plywood;
    MoveL Offs(pOrigin,161.34,-24.55,-0.00),v40,z0,tcp\WObj:=Plywood;
    MoveL Offs(pOrigin,161.34,-22.81,-0.00),v40,z0,tcp\WObj:=Plywood;
    MoveL Offs(pOrigin,161.02,-26.25,-0.00),v40,z0,tcp\WObj:=Plywood;
    MoveL Offs(pOrigin,159.89,-29.01,-0.00),v40,z0,tcp\WObj:=Plywood;
    MoveL Offs(pOrigin,158.75,-30.64,-0.00),v40,fine,tcp\WObj:=Plywood;
    MoveL Offs(pOrigin,158.75,-30.64,-6.00),v60,z5,tcp\WObj:=Plywood;
    MoveL Offs(pOrigin,157.05,-36.56,-6.00),vTravel,z5,tcp\WObj:=Plywood;
    MoveL Offs(pOrigin,157.05,-36.56,-0.00),v60,z0,tcp\WObj:=Plywood;
    MoveL Offs(pOrigin,159.11,-37.51,-0.00),v40,z0,tcp\WObj:=Plywood;
    MoveL Offs(pOrigin,163.57,-38.58,-0.00),v40,z0,tcp\WObj:=Plywood;
    MoveL Offs(pOrigin,176.74,-40.49,-0.00),v40,z0,tcp\WObj:=Plywood;
    MoveL Offs(pOrigin,183.86,-40.70,-0.00),v40,z0,tcp\WObj:=Plywood;
    MoveL Offs(pOrigin,188.01,-39.96,-0.00),v40,z0,tcp\WObj:=Plywood;
    MoveL Offs(pOrigin,190.56,-38.93,-0.00),v40,z0,tcp\WObj:=Plywood;
    MoveL Offs(pOrigin,193.00,-37.41,-0.00),v40,z0,tcp\WObj:=Plywood;
    MoveL Offs(pOrigin,196.93,-33.79,-0.00),v40,z0,tcp\WObj:=Plywood;
    MoveL Offs(pOrigin,199.94,-29.12,-0.00),v40,z0,tcp\WObj:=Plywood;
    MoveL Offs(pOrigin,201.18,-24.41,-0.00),v40,z0,tcp\WObj:=Plywood;
    MoveL Offs(pOrigin,200.76,-27.52,-0.00),v40,z0,tcp\WObj:=Plywood;
    MoveL Offs(pOrigin,199.73,-30.08,-0.00),v40,z0,tcp\WObj:=Plywood;
    MoveL Offs(pOrigin,197.14,-33.90,-0.00),v40,z0,tcp\WObj:=Plywood;
    MoveL Offs(pOrigin,194.38,-36.66,-0.00),v40,z0,tcp\WObj:=Plywood;
    MoveL Offs(pOrigin,191.94,-38.40,-0.00),v40,z0,tcp\WObj:=Plywood;
    MoveL Offs(pOrigin,189.39,-39.67,-0.00),v40,z0,tcp\WObj:=Plywood;
    MoveL Offs(pOrigin,186.31,-40.59,-0.00),v40,z0,tcp\WObj:=Plywood;
    MoveL Offs(pOrigin,181.31,-41.34,-0.00),v40,z0,tcp\WObj:=Plywood;
    MoveL Offs(pOrigin,183.97,-42.97,-0.00),v40,z0,tcp\WObj:=Plywood;
    MoveL Offs(pOrigin,186.94,-44.21,-0.00),v40,z0,tcp\WObj:=Plywood;
    MoveL Offs(pOrigin,189.18,-44.63,-0.00),v40,z0,tcp\WObj:=Plywood;
    MoveL Offs(pOrigin,192.36,-44.31,-0.00),v40,z0,tcp\WObj:=Plywood;
    MoveL Offs(pOrigin,196.82,-42.86,-0.00),v40,z0,tcp\WObj:=Plywood;
    MoveL Offs(pOrigin,200.97,-40.63,-0.00),v40,z0,tcp\WObj:=Plywood;
    MoveL Offs(pOrigin,204.16,-38.26,-0.00),v40,z0,tcp\WObj:=Plywood;
    MoveL Offs(pOrigin,206.74,-35.17,-0.00),v40,z0,tcp\WObj:=Plywood;
    MoveL Offs(pOrigin,207.56,-30.92,-0.00),v40,z0,tcp\WObj:=Plywood;
    MoveL Offs(pOrigin,207.13,-28.06,-0.00),v40,z0,tcp\WObj:=Plywood;
    MoveL Offs(pOrigin,206.21,-25.72,-0.00),v40,z0,tcp\WObj:=Plywood;
    MoveL Offs(pOrigin,205.32,-24.44,-0.00),v40,z0,tcp\WObj:=Plywood;
    MoveL Offs(pOrigin,204.16,-23.52,-0.00),v40,z0,tcp\WObj:=Plywood;
    MoveL Offs(pOrigin,205.11,-26.99,-0.00),v40,z0,tcp\WObj:=Plywood;
    MoveL Offs(pOrigin,205.01,-30.39,-0.00),v40,z0,tcp\WObj:=Plywood;
    MoveL Offs(pOrigin,203.55,-34.86,-0.00),v40,z0,tcp\WObj:=Plywood;
    MoveL Offs(pOrigin,201.57,-38.08,-0.00),v40,z0,tcp\WObj:=Plywood;
    MoveL Offs(pOrigin,203.66,-34.11,-0.00),v40,z0,tcp\WObj:=Plywood;
    MoveL Offs(pOrigin,204.79,-29.86,-0.00),v40,z0,tcp\WObj:=Plywood;
    MoveL Offs(pOrigin,204.58,-25.83,-0.00),v40,z0,tcp\WObj:=Plywood;
    MoveL Offs(pOrigin,203.98,-23.91,-0.00),v40,z0,tcp\WObj:=Plywood;
    MoveL Offs(pOrigin,203.20,-22.81,-0.00),v40,z0,tcp\WObj:=Plywood;
    MoveL Offs(pOrigin,199.80,-21.47,-0.00),v40,z0,tcp\WObj:=Plywood;
    MoveL Offs(pOrigin,196.29,-20.62,-0.00),v40,z0,tcp\WObj:=Plywood;
    MoveL Offs(pOrigin,183.30,-18.81,-0.00),v40,z0,tcp\WObj:=Plywood;
    MoveL Offs(pOrigin,186.09,-20.02,-0.00),v40,z0,tcp\WObj:=Plywood;
    MoveL Offs(pOrigin,191.97,-21.79,-0.00),v40,z0,tcp\WObj:=Plywood;
    MoveL Offs(pOrigin,189.39,-21.36,-0.00),v40,z0,tcp\WObj:=Plywood;
    MoveL Offs(pOrigin,184.07,-19.80,-0.00),v40,z0,tcp\WObj:=Plywood;
    MoveL Offs(pOrigin,175.47,-16.01,-0.00),v40,z0,tcp\WObj:=Plywood;
    MoveL Offs(pOrigin,172.49,-15.20,-0.00),v40,z0,tcp\WObj:=Plywood;
    MoveL Offs(pOrigin,172.39,-15.41,-0.00),v40,z0,tcp\WObj:=Plywood;
    MoveL Offs(pOrigin,173.98,-16.69,-0.00),v40,z0,tcp\WObj:=Plywood;
    MoveL Offs(pOrigin,174.87,-18.07,-0.00),v40,z0,tcp\WObj:=Plywood;
    MoveL Offs(pOrigin,175.47,-19.98,-0.00),v40,z0,tcp\WObj:=Plywood;
    MoveL Offs(pOrigin,175.47,-21.68,-0.00),v40,z0,tcp\WObj:=Plywood;
    MoveL Offs(pOrigin,173.91,-25.72,-0.00),v40,z0,tcp\WObj:=Plywood;
    MoveL Offs(pOrigin,171.54,-29.44,-0.00),v40,z0,tcp\WObj:=Plywood;
    MoveL Offs(pOrigin,167.93,-33.26,-0.00),v40,z0,tcp\WObj:=Plywood;
    MoveL Offs(pOrigin,163.78,-35.85,-0.00),v40,z0,tcp\WObj:=Plywood;
    MoveL Offs(pOrigin,160.91,-36.77,-0.00),v40,z0,tcp\WObj:=Plywood;
    MoveL Offs(pOrigin,157.05,-36.56,-0.00),v40,fine,tcp\WObj:=Plywood;
    MoveL Offs(pOrigin,157.05,-36.56,-6.00),v60,z5,tcp\WObj:=Plywood;
    MoveL Offs(pOrigin,167.46,-31.07,-6.00),vTravel,z5,tcp\WObj:=Plywood;
    MoveL Offs(pOrigin,167.46,-31.07,-0.00),v60,z0,tcp\WObj:=Plywood;
    MoveL Offs(pOrigin,168.99,-28.55,-0.00),v40,z0,tcp\WObj:=Plywood;
  ENDPROC

  PROC DrawPart11()
    MoveL Offs(pOrigin,167.46,-31.07,-0.00),v40,fine,tcp\WObj:=Plywood;
    MoveL Offs(pOrigin,167.46,-31.07,-6.00),v60,z5,tcp\WObj:=Plywood;
    MoveL Offs(pOrigin,170.97,-38.89,-6.00),vTravel,z5,tcp\WObj:=Plywood;
    MoveL Offs(pOrigin,170.97,-38.89,-0.00),v60,z0,tcp\WObj:=Plywood;
    MoveL Offs(pOrigin,176.00,-37.94,-0.00),v40,z0,tcp\WObj:=Plywood;
    MoveL Offs(pOrigin,181.84,-35.85,-0.00),v40,z0,tcp\WObj:=Plywood;
    MoveL Offs(pOrigin,187.26,-32.62,-0.00),v40,z0,tcp\WObj:=Plywood;
    MoveL Offs(pOrigin,191.44,-28.98,-0.00),v40,z0,tcp\WObj:=Plywood;
    MoveL Offs(pOrigin,186.94,-33.16,-0.00),v40,z0,tcp\WObj:=Plywood;
    MoveL Offs(pOrigin,181.63,-36.27,-0.00),v40,z0,tcp\WObj:=Plywood;
    MoveL Offs(pOrigin,175.26,-38.36,-0.00),v40,z0,tcp\WObj:=Plywood;
    MoveL Offs(pOrigin,170.97,-38.89,-0.00),v40,fine,tcp\WObj:=Plywood;
    MoveL Offs(pOrigin,170.97,-38.89,-6.00),v60,z5,tcp\WObj:=Plywood;
    MoveL Offs(pOrigin,169.20,-40.20,-6.00),vTravel,z5,tcp\WObj:=Plywood;
    MoveL Offs(pOrigin,169.20,-40.20,-0.00),v60,z0,tcp\WObj:=Plywood;
    MoveL Offs(pOrigin,171.36,-45.06,-0.00),v40,z0,tcp\WObj:=Plywood;
    MoveL Offs(pOrigin,173.66,-51.57,-0.00),v40,z0,tcp\WObj:=Plywood;
    MoveL Offs(pOrigin,174.41,-49.52,-0.00),v40,z0,tcp\WObj:=Plywood;
    MoveL Offs(pOrigin,173.49,-40.91,-0.00),v40,z0,tcp\WObj:=Plywood;
    MoveL Offs(pOrigin,169.20,-40.20,-0.00),v40,fine,tcp\WObj:=Plywood;
    MoveL Offs(pOrigin,169.20,-40.20,-6.00),v60,z5,tcp\WObj:=Plywood;
    MoveL Offs(pOrigin,174.41,-40.84,-6.00),vTravel,z5,tcp\WObj:=Plywood;
    MoveL Offs(pOrigin,174.41,-40.84,-0.00),v60,z0,tcp\WObj:=Plywood;
    MoveL Offs(pOrigin,175.15,-48.17,-0.00),v40,z0,tcp\WObj:=Plywood;
    MoveL Offs(pOrigin,175.79,-46.65,-0.00),v40,z0,tcp\WObj:=Plywood;
    MoveL Offs(pOrigin,176.32,-41.34,-0.00),v40,z0,tcp\WObj:=Plywood;
    MoveL Offs(pOrigin,176.00,-41.02,-0.00),v40,z0,tcp\WObj:=Plywood;
    MoveL Offs(pOrigin,174.41,-40.84,-0.00),v40,fine,tcp\WObj:=Plywood;
    MoveL Offs(pOrigin,174.41,-40.84,-6.00),v60,z5,tcp\WObj:=Plywood;
    MoveL Offs(pOrigin,177.10,-41.34,-6.00),vTravel,z5,tcp\WObj:=Plywood;
    MoveL Offs(pOrigin,177.10,-41.34,-0.00),v60,z0,tcp\WObj:=Plywood;
    MoveL Offs(pOrigin,176.64,-43.78,-0.00),v40,z0,tcp\WObj:=Plywood;
    MoveL Offs(pOrigin,176.53,-47.50,-0.00),v40,z0,tcp\WObj:=Plywood;
    MoveL Offs(pOrigin,177.13,-50.26,-0.00),v40,z0,tcp\WObj:=Plywood;
    MoveL Offs(pOrigin,178.30,-52.53,-0.00),v40,z0,tcp\WObj:=Plywood;
    MoveL Offs(pOrigin,176.92,-50.37,-0.00),v40,z0,tcp\WObj:=Plywood;
    MoveL Offs(pOrigin,176.21,-48.07,-0.00),v40,z0,tcp\WObj:=Plywood;
    MoveL Offs(pOrigin,174.41,-51.54,-0.00),v40,z0,tcp\WObj:=Plywood;
    MoveL Offs(pOrigin,175.04,-53.03,-0.00),v40,z0,tcp\WObj:=Plywood;
    MoveL Offs(pOrigin,178.12,-56.00,-0.00),v40,z0,tcp\WObj:=Plywood;
    MoveL Offs(pOrigin,182.59,-58.90,-0.00),v40,z0,tcp\WObj:=Plywood;
    MoveL Offs(pOrigin,189.92,-62.62,-0.00),v40,z0,tcp\WObj:=Plywood;
    MoveL Offs(pOrigin,193.57,-64.07,-0.00),v40,z0,tcp\WObj:=Plywood;
    MoveL Offs(pOrigin,189.28,-62.62,-0.00),v40,z0,tcp\WObj:=Plywood;
    MoveL Offs(pOrigin,183.12,-59.54,-0.00),v40,z0,tcp\WObj:=Plywood;
    MoveL Offs(pOrigin,178.76,-56.96,-0.00),v40,z0,tcp\WObj:=Plywood;
    MoveL Offs(pOrigin,174.73,-53.77,-0.00),v40,z0,tcp\WObj:=Plywood;
    MoveL Offs(pOrigin,175.01,-55.36,-0.00),v40,z0,tcp\WObj:=Plywood;
    MoveL Offs(pOrigin,177.06,-57.70,-0.00),v40,z0,tcp\WObj:=Plywood;
    MoveL Offs(pOrigin,179.82,-59.65,-0.00),v40,z0,tcp\WObj:=Plywood;
    MoveL Offs(pOrigin,184.11,-61.63,-0.00),v40,z0,tcp\WObj:=Plywood;
    MoveL Offs(pOrigin,178.87,-59.54,-0.00),v40,z0,tcp\WObj:=Plywood;
    MoveL Offs(pOrigin,175.15,-56.67,-0.00),v40,z0,tcp\WObj:=Plywood;
    MoveL Offs(pOrigin,176.07,-58.66,-0.00),v40,z0,tcp\WObj:=Plywood;
    MoveL Offs(pOrigin,179.08,-62.69,-0.00),v40,z0,tcp\WObj:=Plywood;
    MoveL Offs(pOrigin,183.58,-66.48,-0.00),v40,z0,tcp\WObj:=Plywood;
    MoveL Offs(pOrigin,181.10,-64.93,-0.00),v40,z0,tcp\WObj:=Plywood;
    MoveL Offs(pOrigin,178.23,-62.27,-0.00),v40,z0,tcp\WObj:=Plywood;
    MoveL Offs(pOrigin,175.04,-57.56,-0.00),v40,z0,tcp\WObj:=Plywood;
    MoveL Offs(pOrigin,175.86,-61.74,-0.00),v40,z0,tcp\WObj:=Plywood;
    MoveL Offs(pOrigin,177.98,-65.99,-0.00),v40,z0,tcp\WObj:=Plywood;
    MoveL Offs(pOrigin,180.04,-68.75,-0.00),v40,z0,tcp\WObj:=Plywood;
    MoveL Offs(pOrigin,182.91,-71.51,-0.00),v40,z0,tcp\WObj:=Plywood;
    MoveL Offs(pOrigin,185.77,-73.35,-0.00),v40,z0,tcp\WObj:=Plywood;
    MoveL Offs(pOrigin,188.36,-74.45,-0.00),v40,z0,tcp\WObj:=Plywood;
    MoveL Offs(pOrigin,184.93,-73.35,-0.00),v40,z0,tcp\WObj:=Plywood;
    MoveL Offs(pOrigin,181.52,-71.09,-0.00),v40,z0,tcp\WObj:=Plywood;
    MoveL Offs(pOrigin,179.29,-68.86,-0.00),v40,z0,tcp\WObj:=Plywood;
    MoveL Offs(pOrigin,176.14,-64.50,-0.00),v40,z0,tcp\WObj:=Plywood;
    MoveL Offs(pOrigin,177.13,-67.26,-0.00),v40,z0,tcp\WObj:=Plywood;
    MoveL Offs(pOrigin,179.61,-70.66,-0.00),v40,z0,tcp\WObj:=Plywood;
    MoveL Offs(pOrigin,183.54,-74.70,-0.00),v40,z0,tcp\WObj:=Plywood;
    MoveL Offs(pOrigin,187.44,-77.78,-0.00),v40,z0,tcp\WObj:=Plywood;
    MoveL Offs(pOrigin,185.56,-76.72,-0.00),v40,z0,tcp\WObj:=Plywood;
    MoveL Offs(pOrigin,182.48,-74.28,-0.00),v40,z0,tcp\WObj:=Plywood;
    MoveL Offs(pOrigin,178.98,-70.56,-0.00),v40,z0,tcp\WObj:=Plywood;
    MoveL Offs(pOrigin,176.67,-67.26,-0.00),v40,z0,tcp\WObj:=Plywood;
    MoveL Offs(pOrigin,178.55,-76.08,-0.00),v40,z0,tcp\WObj:=Plywood;
    MoveL Offs(pOrigin,181.95,-88.72,-0.00),v40,z0,tcp\WObj:=Plywood;
    MoveL Offs(pOrigin,184.04,-94.68,-0.00),v40,z0,tcp\WObj:=Plywood;
    MoveL Offs(pOrigin,185.67,-97.08,-0.00),v40,z0,tcp\WObj:=Plywood;
    MoveL Offs(pOrigin,186.84,-96.84,-0.00),v40,z0,tcp\WObj:=Plywood;
    MoveL Offs(pOrigin,187.86,-95.63,-0.00),v40,z0,tcp\WObj:=Plywood;
    MoveL Offs(pOrigin,186.16,-92.12,-0.00),v40,z0,tcp\WObj:=Plywood;
    MoveL Offs(pOrigin,185.14,-89.11,-0.00),v40,z0,tcp\WObj:=Plywood;
    MoveL Offs(pOrigin,188.11,-95.17,-0.00),v40,z0,tcp\WObj:=Plywood;
    MoveL Offs(pOrigin,190.13,-87.45,-0.00),v40,z0,tcp\WObj:=Plywood;
    MoveL Offs(pOrigin,189.74,-86.28,-0.00),v40,z0,tcp\WObj:=Plywood;
    MoveL Offs(pOrigin,188.11,-83.84,-0.00),v40,z0,tcp\WObj:=Plywood;
    MoveL Offs(pOrigin,180.00,-73.28,-0.00),v40,z0,tcp\WObj:=Plywood;
    MoveL Offs(pOrigin,189.71,-84.65,-0.00),v40,z0,tcp\WObj:=Plywood;
    MoveL Offs(pOrigin,192.50,-77.99,-0.00),v40,z0,tcp\WObj:=Plywood;
    MoveL Offs(pOrigin,192.79,-75.97,-0.00),v40,z0,tcp\WObj:=Plywood;
    MoveL Offs(pOrigin,191.51,-74.28,-0.00),v40,z0,tcp\WObj:=Plywood;
    MoveL Offs(pOrigin,186.59,-69.88,-0.00),v40,z0,tcp\WObj:=Plywood;
    MoveL Offs(pOrigin,192.47,-74.28,-0.00),v40,z0,tcp\WObj:=Plywood;
    MoveL Offs(pOrigin,194.31,-72.47,-0.00),v40,z0,tcp\WObj:=Plywood;
    MoveL Offs(pOrigin,195.09,-66.41,-0.00),v40,z0,tcp\WObj:=Plywood;
    MoveL Offs(pOrigin,189.78,-64.82,-0.00),v40,z0,tcp\WObj:=Plywood;
    MoveL Offs(pOrigin,195.76,-65.99,-0.00),v40,z0,tcp\WObj:=Plywood;
    MoveL Offs(pOrigin,196.93,-65.99,-0.00),v40,z0,tcp\WObj:=Plywood;
    MoveL Offs(pOrigin,197.50,-65.56,-0.00),v40,z0,tcp\WObj:=Plywood;
    MoveL Offs(pOrigin,197.57,-61.84,-0.00),v40,z0,tcp\WObj:=Plywood;
    MoveL Offs(pOrigin,199.52,-58.34,-0.00),v40,z0,tcp\WObj:=Plywood;
    MoveL Offs(pOrigin,200.08,-56.00,-0.00),v40,z0,tcp\WObj:=Plywood;
    MoveL Offs(pOrigin,195.98,-58.16,-0.00),v40,z0,tcp\WObj:=Plywood;
    MoveL Offs(pOrigin,193.74,-58.87,-0.00),v40,z0,tcp\WObj:=Plywood;
    MoveL Offs(pOrigin,191.80,-59.08,-0.00),v40,z0,tcp\WObj:=Plywood;
    MoveL Offs(pOrigin,195.12,-58.16,-0.00),v40,z0,tcp\WObj:=Plywood;
    MoveL Offs(pOrigin,198.21,-56.57,-0.00),v40,z0,tcp\WObj:=Plywood;
    MoveL Offs(pOrigin,200.23,-55.04,-0.00),v40,z0,tcp\WObj:=Plywood;
    MoveL Offs(pOrigin,202.17,-52.71,-0.00),v40,z0,tcp\WObj:=Plywood;
    MoveL Offs(pOrigin,203.62,-49.09,-0.00),v40,z0,tcp\WObj:=Plywood;
    MoveL Offs(pOrigin,205.29,-42.83,-0.00),v40,z0,tcp\WObj:=Plywood;
    MoveL Offs(pOrigin,206.92,-38.79,-0.00),v40,z0,tcp\WObj:=Plywood;
    MoveL Offs(pOrigin,207.13,-35.99,-0.00),v40,z0,tcp\WObj:=Plywood;
    MoveL Offs(pOrigin,204.69,-38.58,-0.00),v40,z0,tcp\WObj:=Plywood;
    MoveL Offs(pOrigin,200.33,-41.59,-0.00),v40,z0,tcp\WObj:=Plywood;
    MoveL Offs(pOrigin,195.12,-44.03,-0.00),v40,z0,tcp\WObj:=Plywood;
    MoveL Offs(pOrigin,191.48,-45.06,-0.00),v40,z0,tcp\WObj:=Plywood;
  ENDPROC

